// SIMATIC S7-200 project (STEP 7-Micro/WIN), CPU 224 CN REL 02.01

// OB1: protected block, not included

SUBROUTINE_BLOCK PIDCALCULATE:SBR0
TITLE=子程序注释
BEGIN
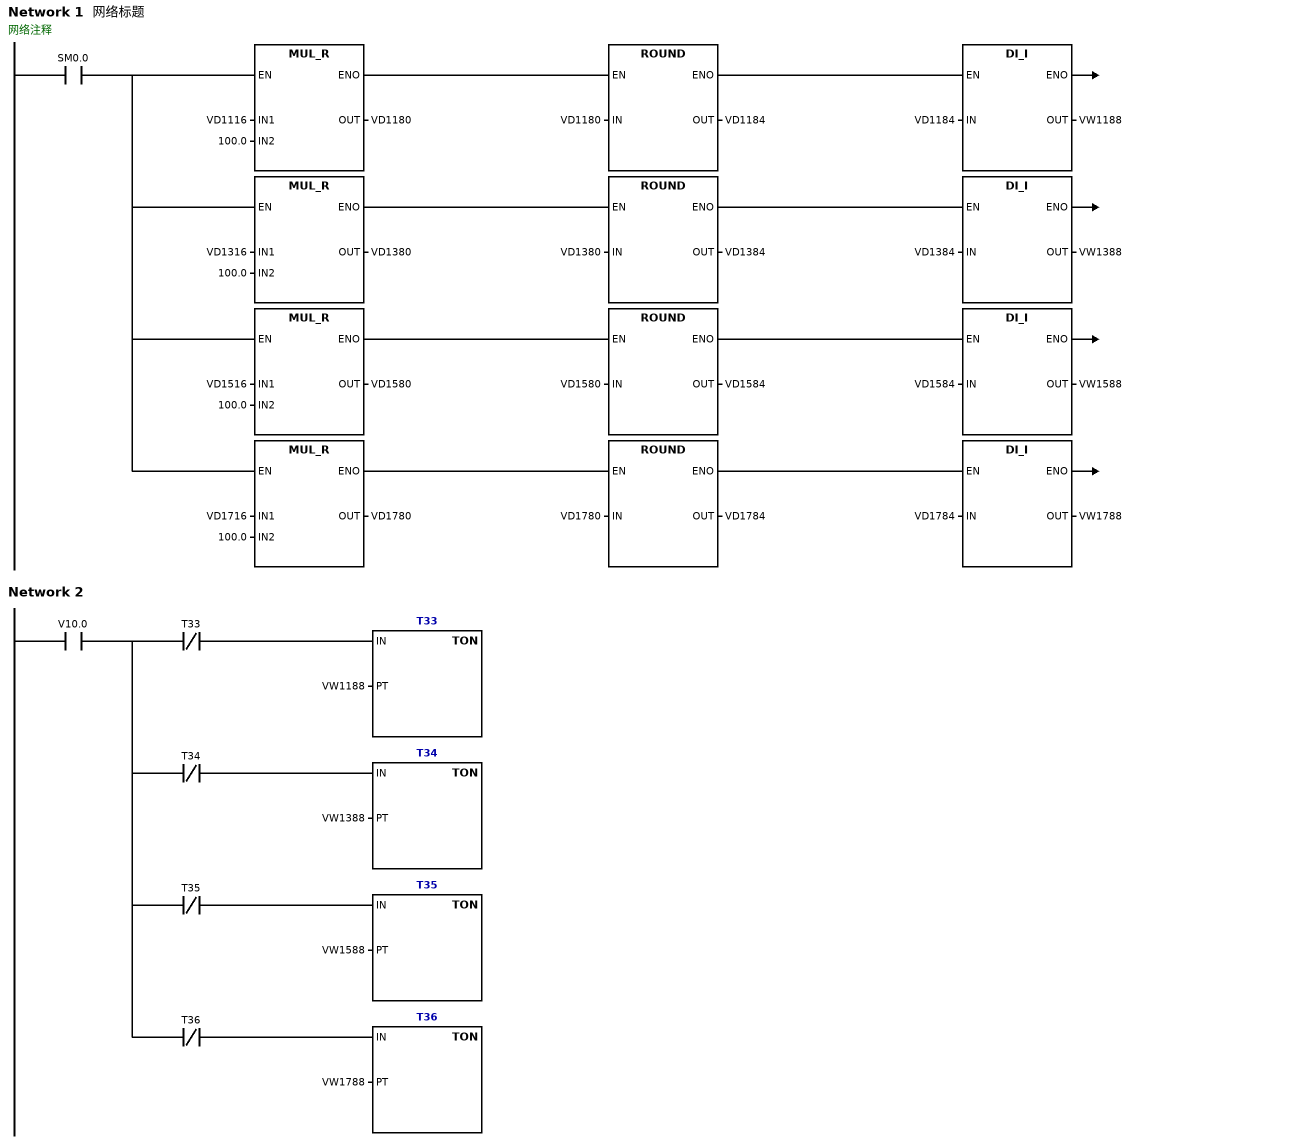
Network 1 // 网络标题
// 网络注释
LD     SM0.0
LPS
MOVR   VD1116, VD1180
AENO
*R     100.0, VD1180
AENO
ROUND  VD1180, VD1184
AENO
DTI    VD1184, VW1188
LRD
MOVR   VD1316, VD1380
AENO
*R     100.0, VD1380
AENO
ROUND  VD1380, VD1384
AENO
DTI    VD1384, VW1388
LRD
MOVR   VD1516, VD1580
AENO
*R     100.0, VD1580
AENO
ROUND  VD1580, VD1584
AENO
DTI    VD1584, VW1588
LPP
MOVR   VD1716, VD1780
AENO
*R     100.0, VD1780
AENO
ROUND  VD1780, VD1784
AENO
DTI    VD1784, VW1788
Network 2
LD     V10.0
LPS
AN     T33
TON    T33, VW1188
LRD
AN     T34
TON    T34, VW1388
LRD
AN     T35
TON    T35, VW1588
LPP
AN     T36
TON    T36, VW1788
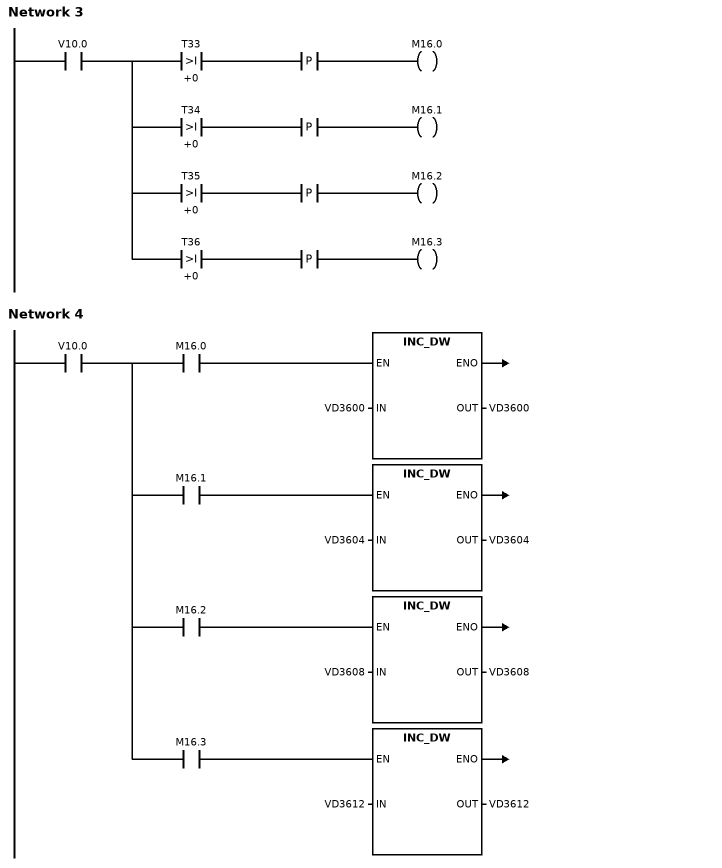
Network 3
LD     V10.0
LPS
AW>    T33, +0
EU
=      M16.0
LRD
AW>    T34, +0
EU
=      M16.1
LRD
AW>    T35, +0
EU
=      M16.2
LPP
AW>    T36, +0
EU
=      M16.3
Network 4
LD     V10.0
LPS
A      M16.0
INCD   VD3600
LRD
A      M16.1
INCD   VD3604
LRD
A      M16.2
INCD   VD3608
LPP
A      M16.3
INCD   VD3612
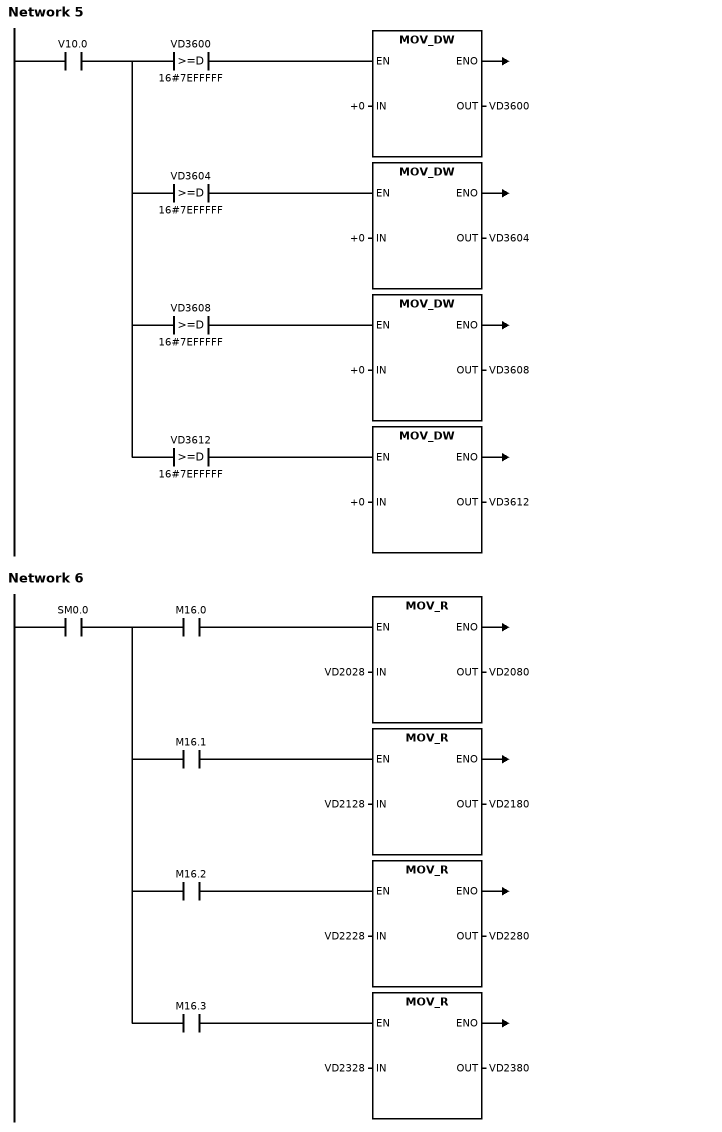
Network 5
LD     V10.0
LPS
AD>=   VD3600, 16#7EFFFFF
MOVD   +0, VD3600
LRD
AD>=   VD3604, 16#7EFFFFF
MOVD   +0, VD3604
LRD
AD>=   VD3608, 16#7EFFFFF
MOVD   +0, VD3608
LPP
AD>=   VD3612, 16#7EFFFFF
MOVD   +0, VD3612
Network 6
LD     SM0.0
LPS
A      M16.0
MOVR   VD2028, VD2080
LRD
A      M16.1
MOVR   VD2128, VD2180
LRD
A      M16.2
MOVR   VD2228, VD2280
LPP
A      M16.3
MOVR   VD2328, VD2380
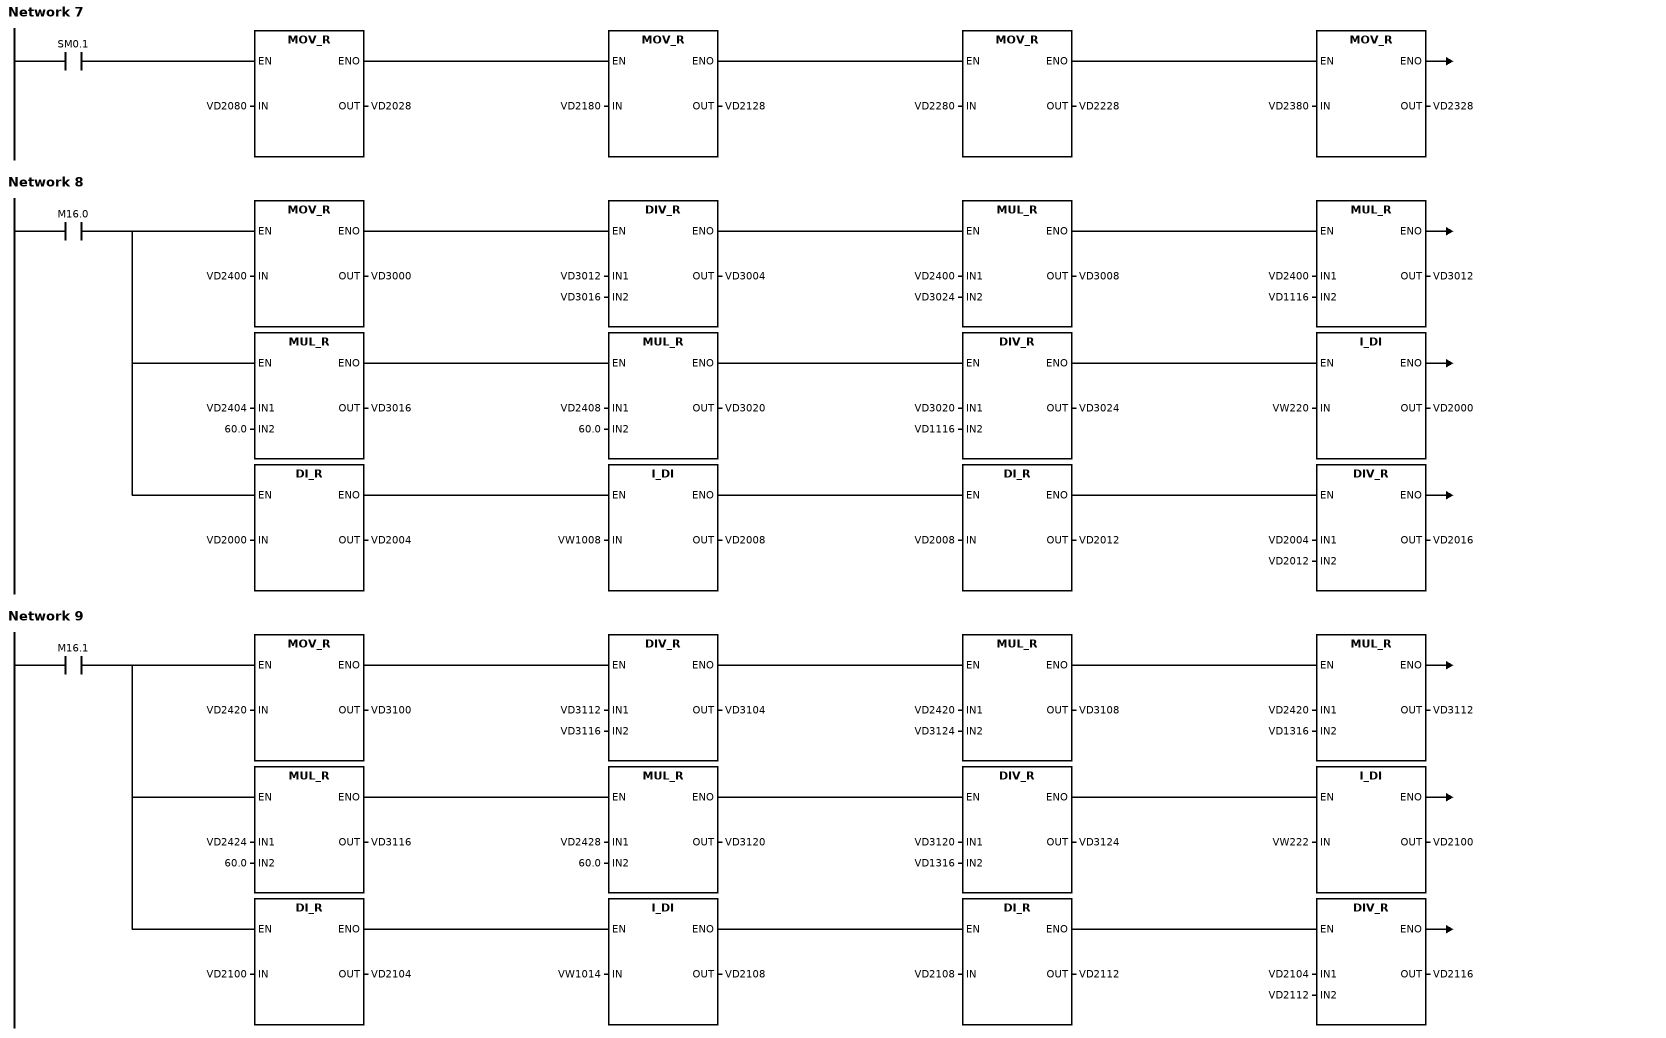
Network 7
LD     SM0.1
MOVR   VD2080, VD2028
AENO
MOVR   VD2180, VD2128
AENO
MOVR   VD2280, VD2228
AENO
MOVR   VD2380, VD2328
Network 8
LD     M16.0
LPS
MOVR   VD2400, VD3000
AENO
MOVR   VD3012, VD3004
AENO
/R     VD3016, VD3004
AENO
MOVR   VD2400, VD3008
AENO
*R     VD3024, VD3008
AENO
MOVR   VD2400, VD3012
*R     VD1116, VD3012
LRD
MOVR   VD2404, VD3016
AENO
*R     60.0, VD3016
AENO
MOVR   VD2408, VD3020
AENO
*R     60.0, VD3020
AENO
MOVR   VD3020, VD3024
AENO
/R     VD1116, VD3024
AENO
ITD    VW220, VD2000
LPP
DTR    VD2000, VD2004
AENO
ITD    VW1008, VD2008
AENO
DTR    VD2008, VD2012
AENO
MOVR   VD2004, VD2016
/R     VD2012, VD2016
Network 9
LD     M16.1
LPS
MOVR   VD2420, VD3100
AENO
MOVR   VD3112, VD3104
AENO
/R     VD3116, VD3104
AENO
MOVR   VD2420, VD3108
AENO
*R     VD3124, VD3108
AENO
MOVR   VD2420, VD3112
*R     VD1316, VD3112
LRD
MOVR   VD2424, VD3116
AENO
*R     60.0, VD3116
AENO
MOVR   VD2428, VD3120
AENO
*R     60.0, VD3120
AENO
MOVR   VD3120, VD3124
AENO
/R     VD1316, VD3124
AENO
ITD    VW222, VD2100
LPP
DTR    VD2100, VD2104
AENO
ITD    VW1014, VD2108
AENO
DTR    VD2108, VD2112
AENO
MOVR   VD2104, VD2116
/R     VD2112, VD2116
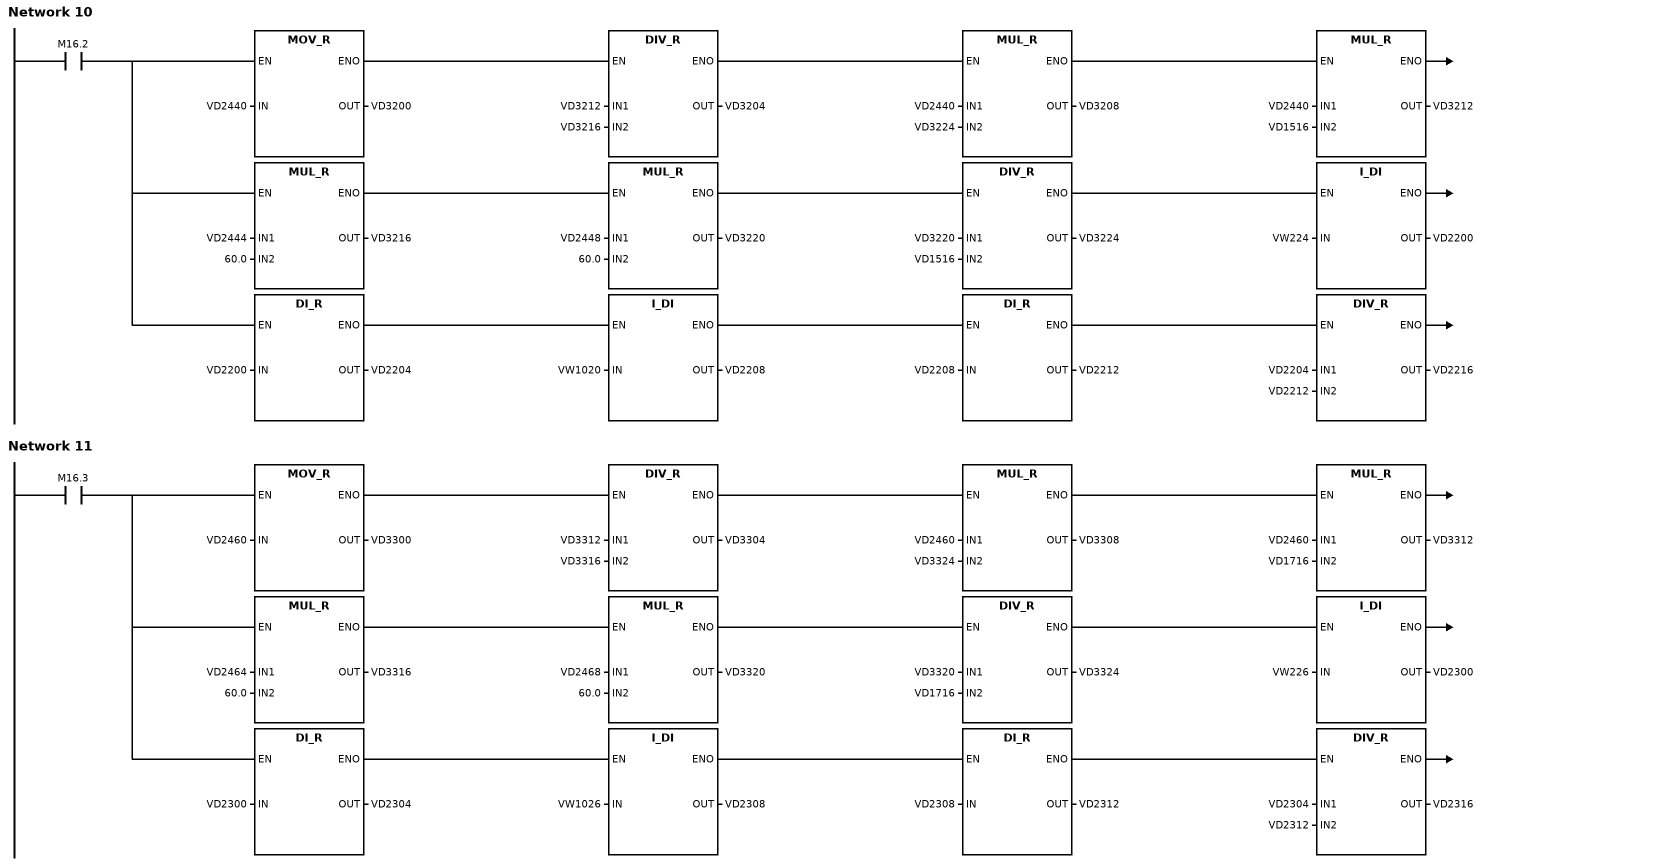
Network 10
LD     M16.2
LPS
MOVR   VD2440, VD3200
AENO
MOVR   VD3212, VD3204
AENO
/R     VD3216, VD3204
AENO
MOVR   VD2440, VD3208
AENO
*R     VD3224, VD3208
AENO
MOVR   VD2440, VD3212
*R     VD1516, VD3212
LRD
MOVR   VD2444, VD3216
AENO
*R     60.0, VD3216
AENO
MOVR   VD2448, VD3220
AENO
*R     60.0, VD3220
AENO
MOVR   VD3220, VD3224
AENO
/R     VD1516, VD3224
AENO
ITD    VW224, VD2200
LPP
DTR    VD2200, VD2204
AENO
ITD    VW1020, VD2208
AENO
DTR    VD2208, VD2212
AENO
MOVR   VD2204, VD2216
/R     VD2212, VD2216
Network 11
LD     M16.3
LPS
MOVR   VD2460, VD3300
AENO
MOVR   VD3312, VD3304
AENO
/R     VD3316, VD3304
AENO
MOVR   VD2460, VD3308
AENO
*R     VD3324, VD3308
AENO
MOVR   VD2460, VD3312
*R     VD1716, VD3312
LRD
MOVR   VD2464, VD3316
AENO
*R     60.0, VD3316
AENO
MOVR   VD2468, VD3320
AENO
*R     60.0, VD3320
AENO
MOVR   VD3320, VD3324
AENO
/R     VD1716, VD3324
AENO
ITD    VW226, VD2300
LPP
DTR    VD2300, VD2304
AENO
ITD    VW1026, VD2308
AENO
DTR    VD2308, VD2312
AENO
MOVR   VD2304, VD2316
/R     VD2312, VD2316
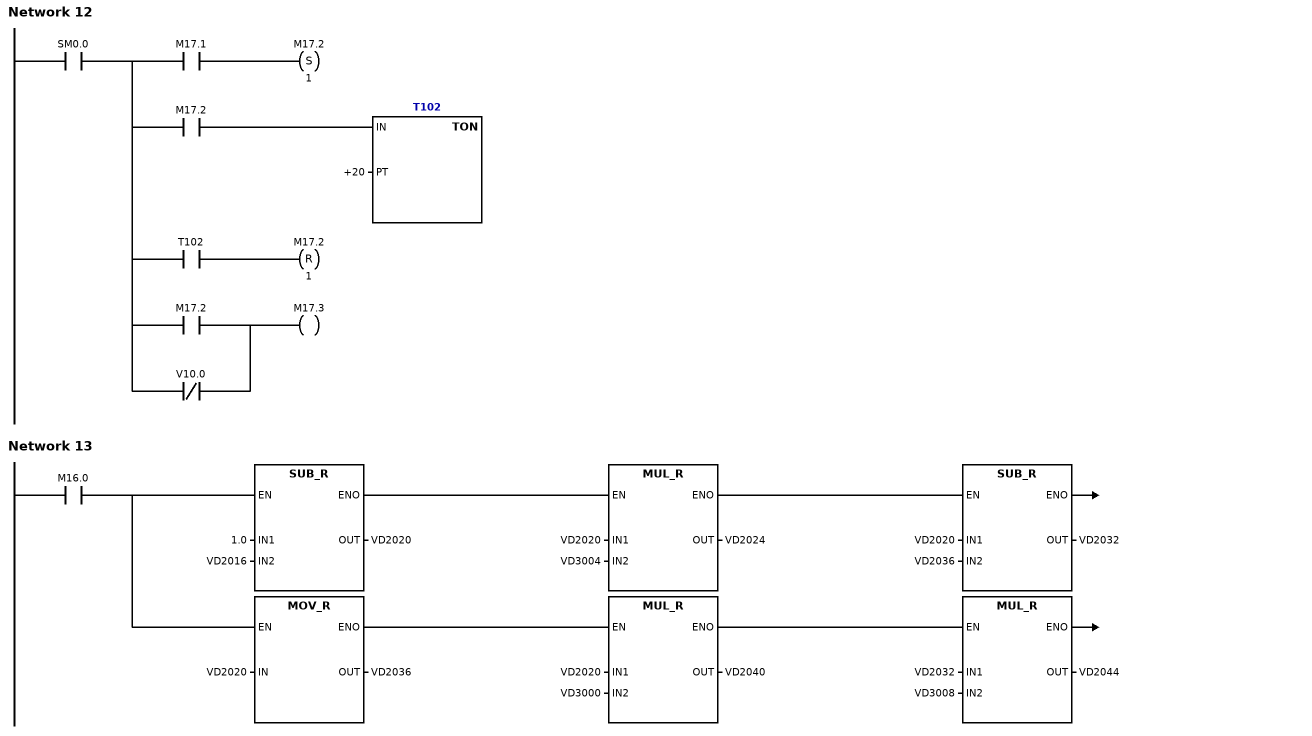
Network 12
LD     SM0.0
LPS
A      M17.1
S      M17.2, 1
LRD
A      M17.2
TON    T102, +20
LRD
A      T102
R      M17.2, 1
LPP
LD     M17.2
ON     V10.0
ALD
=      M17.3
Network 13
LD     M16.0
LPS
MOVR   1.0, VD2020
AENO
-R     VD2016, VD2020
AENO
MOVR   VD2020, VD2024
AENO
*R     VD3004, VD2024
AENO
MOVR   VD2020, VD2032
-R     VD2036, VD2032
LPP
MOVR   VD2020, VD2036
AENO
MOVR   VD2020, VD2040
AENO
*R     VD3000, VD2040
AENO
MOVR   VD2032, VD2044
*R     VD3008, VD2044
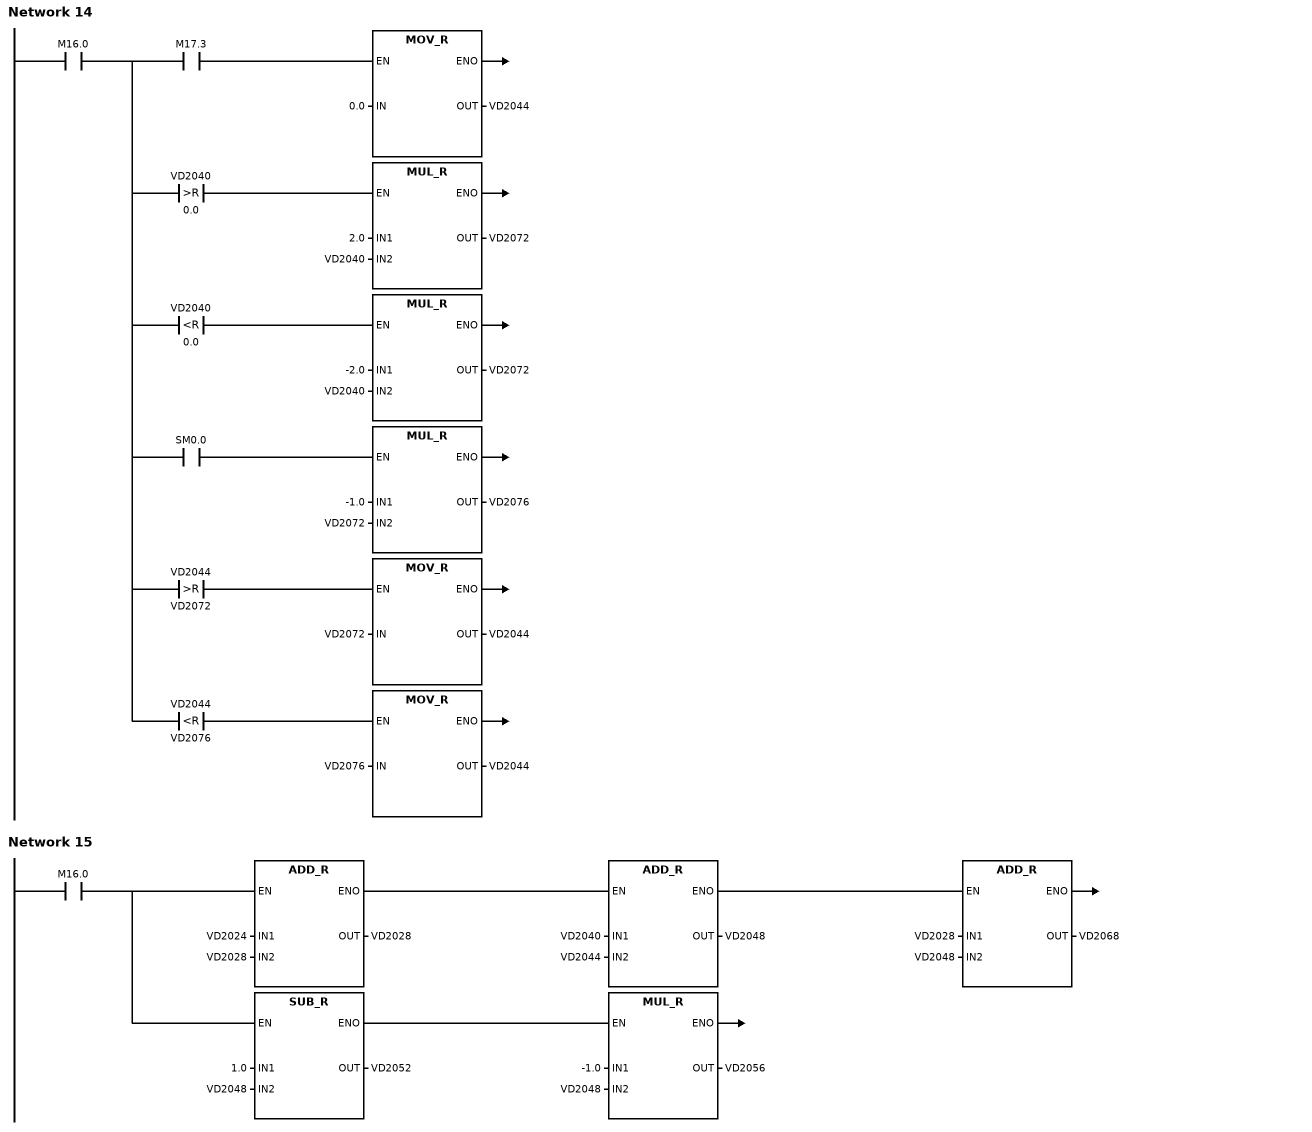
Network 14
LD     M16.0
LPS
A      M17.3
MOVR   0.0, VD2044
LRD
AR>    VD2040, 0.0
MOVR   2.0, VD2072
*R     VD2040, VD2072
LRD
AR<    VD2040, 0.0
MOVR   -2.0, VD2072
*R     VD2040, VD2072
LRD
A      SM0.0
MOVR   -1.0, VD2076
*R     VD2072, VD2076
LRD
AR>    VD2044, VD2072
MOVR   VD2072, VD2044
LPP
AR<    VD2044, VD2076
MOVR   VD2076, VD2044
Network 15
LD     M16.0
LPS
+R     VD2024, VD2028
AENO
MOVR   VD2040, VD2048
AENO
+R     VD2044, VD2048
AENO
MOVR   VD2028, VD2068
+R     VD2048, VD2068
LPP
MOVR   1.0, VD2052
AENO
-R     VD2048, VD2052
AENO
MOVR   -1.0, VD2056
*R     VD2048, VD2056
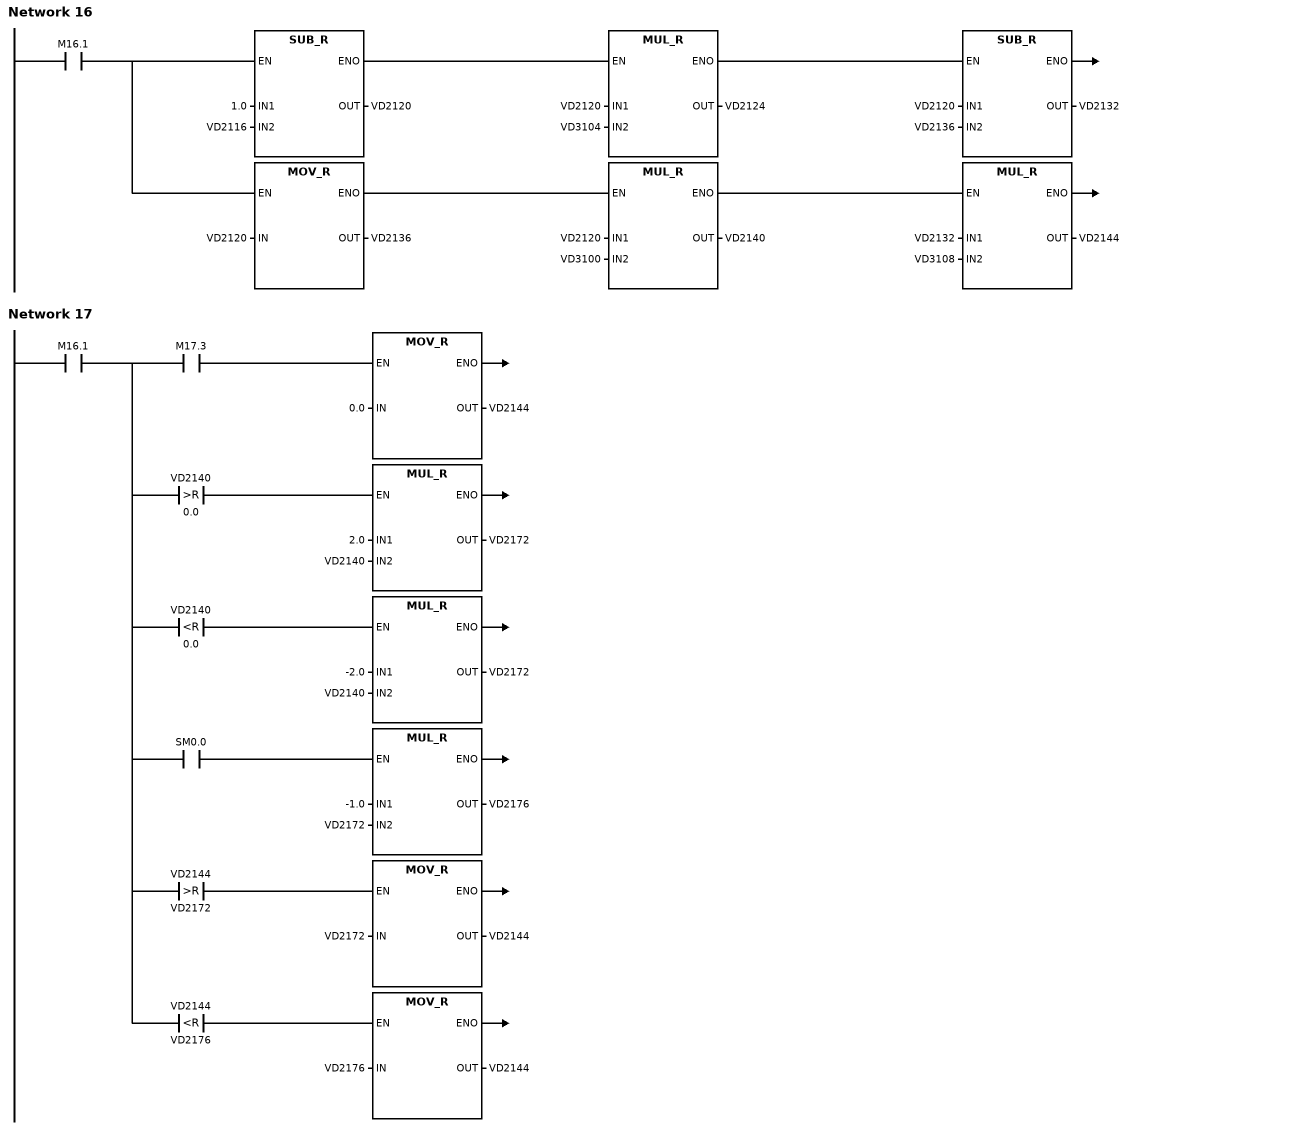
Network 16
LD     M16.1
LPS
MOVR   1.0, VD2120
AENO
-R     VD2116, VD2120
AENO
MOVR   VD2120, VD2124
AENO
*R     VD3104, VD2124
AENO
MOVR   VD2120, VD2132
-R     VD2136, VD2132
LPP
MOVR   VD2120, VD2136
AENO
MOVR   VD2120, VD2140
AENO
*R     VD3100, VD2140
AENO
MOVR   VD2132, VD2144
*R     VD3108, VD2144
Network 17
LD     M16.1
LPS
A      M17.3
MOVR   0.0, VD2144
LRD
AR>    VD2140, 0.0
MOVR   2.0, VD2172
*R     VD2140, VD2172
LRD
AR<    VD2140, 0.0
MOVR   -2.0, VD2172
*R     VD2140, VD2172
LRD
A      SM0.0
MOVR   -1.0, VD2176
*R     VD2172, VD2176
LRD
AR>    VD2144, VD2172
MOVR   VD2172, VD2144
LPP
AR<    VD2144, VD2176
MOVR   VD2176, VD2144
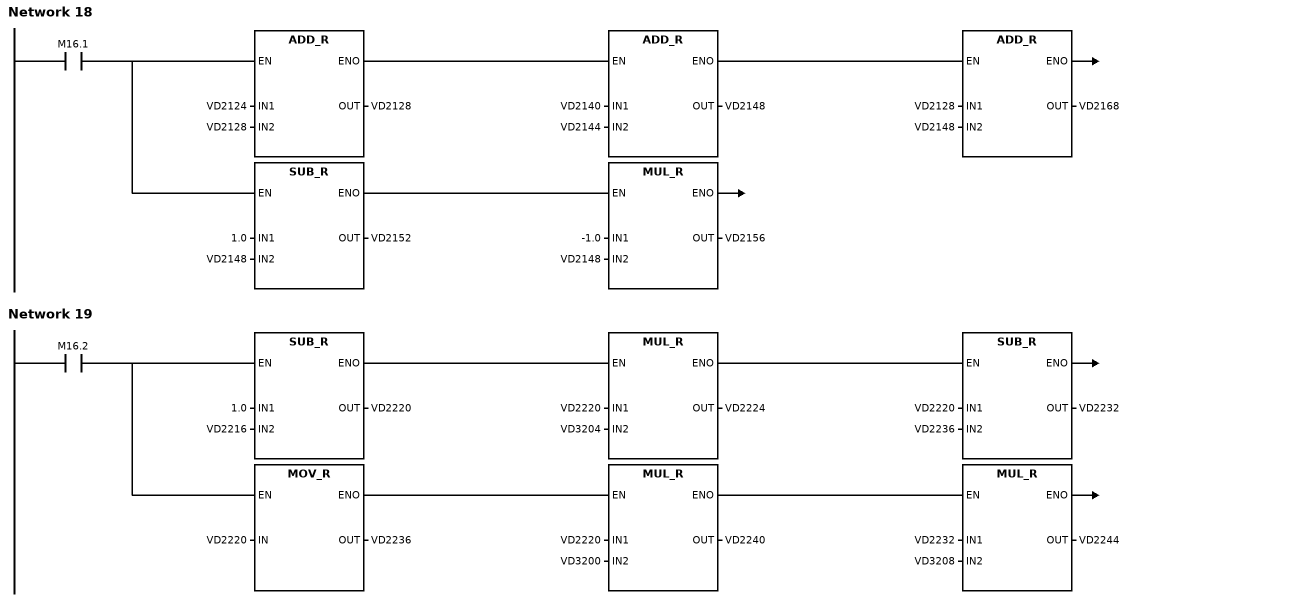
Network 18
LD     M16.1
LPS
+R     VD2124, VD2128
AENO
MOVR   VD2140, VD2148
AENO
+R     VD2144, VD2148
AENO
MOVR   VD2128, VD2168
+R     VD2148, VD2168
LPP
MOVR   1.0, VD2152
AENO
-R     VD2148, VD2152
AENO
MOVR   -1.0, VD2156
*R     VD2148, VD2156
Network 19
LD     M16.2
LPS
MOVR   1.0, VD2220
AENO
-R     VD2216, VD2220
AENO
MOVR   VD2220, VD2224
AENO
*R     VD3204, VD2224
AENO
MOVR   VD2220, VD2232
-R     VD2236, VD2232
LPP
MOVR   VD2220, VD2236
AENO
MOVR   VD2220, VD2240
AENO
*R     VD3200, VD2240
AENO
MOVR   VD2232, VD2244
*R     VD3208, VD2244
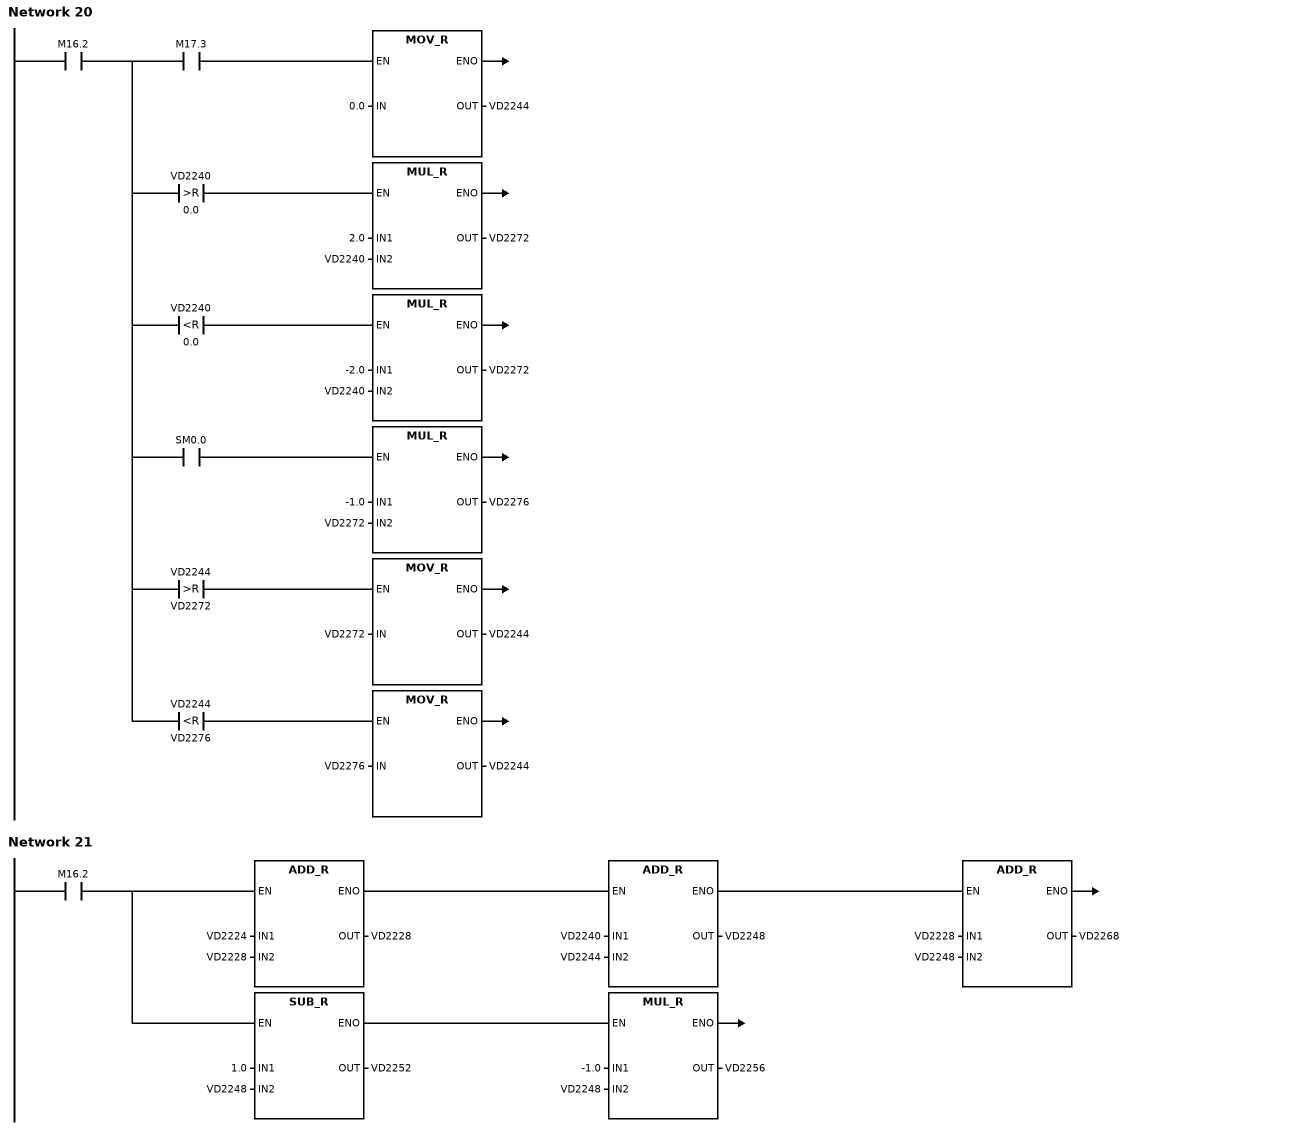
Network 20
LD     M16.2
LPS
A      M17.3
MOVR   0.0, VD2244
LRD
AR>    VD2240, 0.0
MOVR   2.0, VD2272
*R     VD2240, VD2272
LRD
AR<    VD2240, 0.0
MOVR   -2.0, VD2272
*R     VD2240, VD2272
LRD
A      SM0.0
MOVR   -1.0, VD2276
*R     VD2272, VD2276
LRD
AR>    VD2244, VD2272
MOVR   VD2272, VD2244
LPP
AR<    VD2244, VD2276
MOVR   VD2276, VD2244
Network 21
LD     M16.2
LPS
+R     VD2224, VD2228
AENO
MOVR   VD2240, VD2248
AENO
+R     VD2244, VD2248
AENO
MOVR   VD2228, VD2268
+R     VD2248, VD2268
LPP
MOVR   1.0, VD2252
AENO
-R     VD2248, VD2252
AENO
MOVR   -1.0, VD2256
*R     VD2248, VD2256
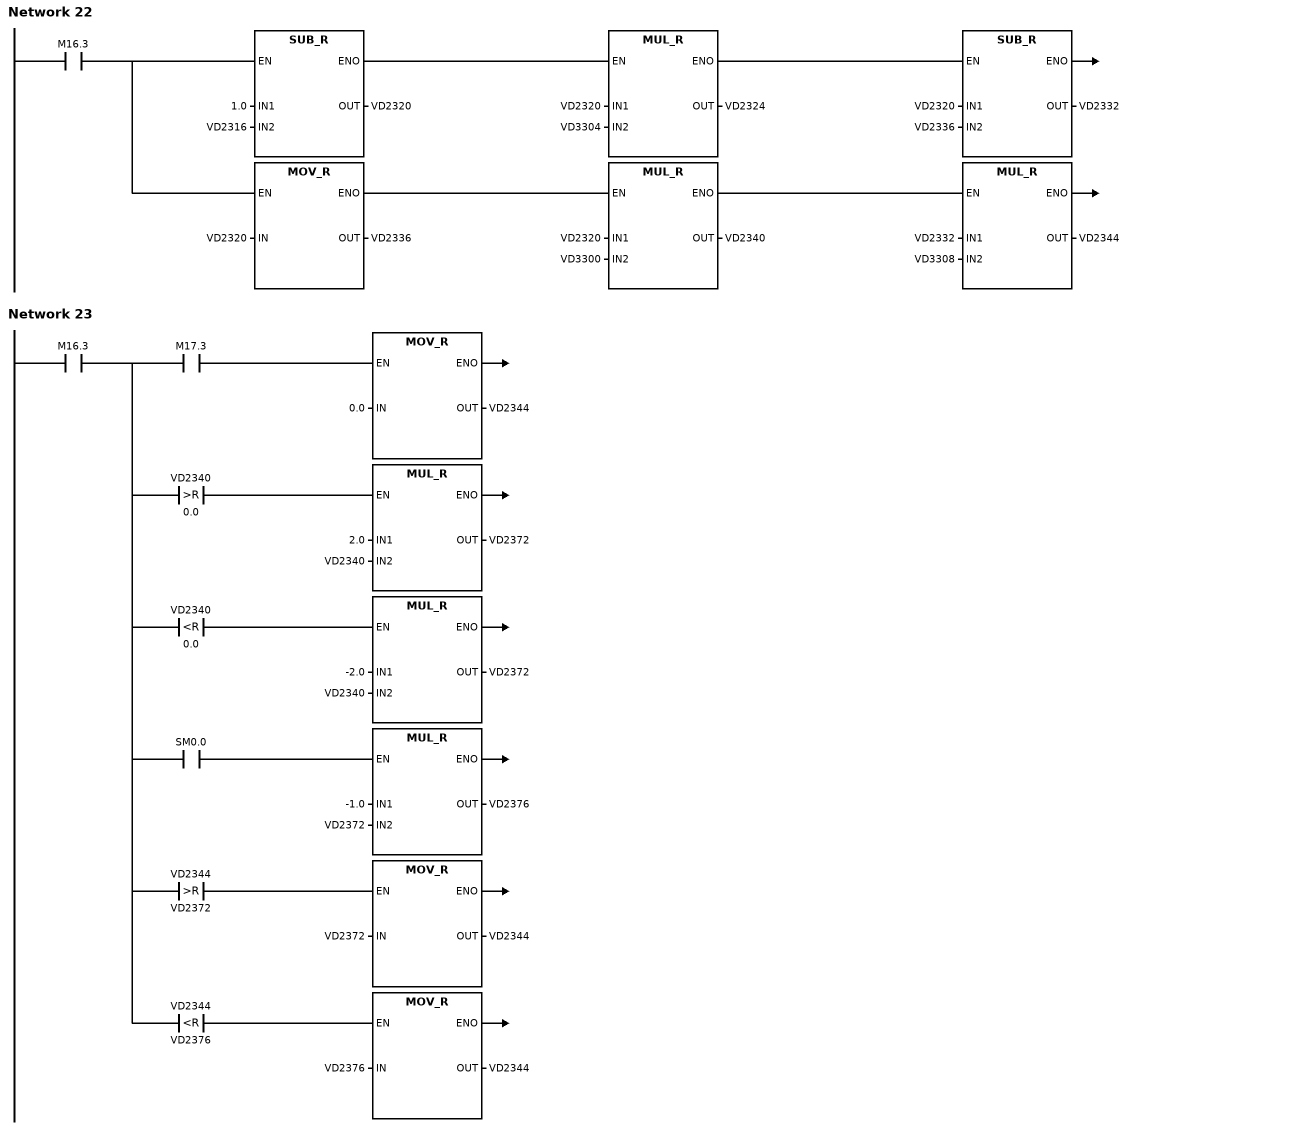
Network 22
LD     M16.3
LPS
MOVR   1.0, VD2320
AENO
-R     VD2316, VD2320
AENO
MOVR   VD2320, VD2324
AENO
*R     VD3304, VD2324
AENO
MOVR   VD2320, VD2332
-R     VD2336, VD2332
LPP
MOVR   VD2320, VD2336
AENO
MOVR   VD2320, VD2340
AENO
*R     VD3300, VD2340
AENO
MOVR   VD2332, VD2344
*R     VD3308, VD2344
Network 23
LD     M16.3
LPS
A      M17.3
MOVR   0.0, VD2344
LRD
AR>    VD2340, 0.0
MOVR   2.0, VD2372
*R     VD2340, VD2372
LRD
AR<    VD2340, 0.0
MOVR   -2.0, VD2372
*R     VD2340, VD2372
LRD
A      SM0.0
MOVR   -1.0, VD2376
*R     VD2372, VD2376
LRD
AR>    VD2344, VD2372
MOVR   VD2372, VD2344
LPP
AR<    VD2344, VD2376
MOVR   VD2376, VD2344
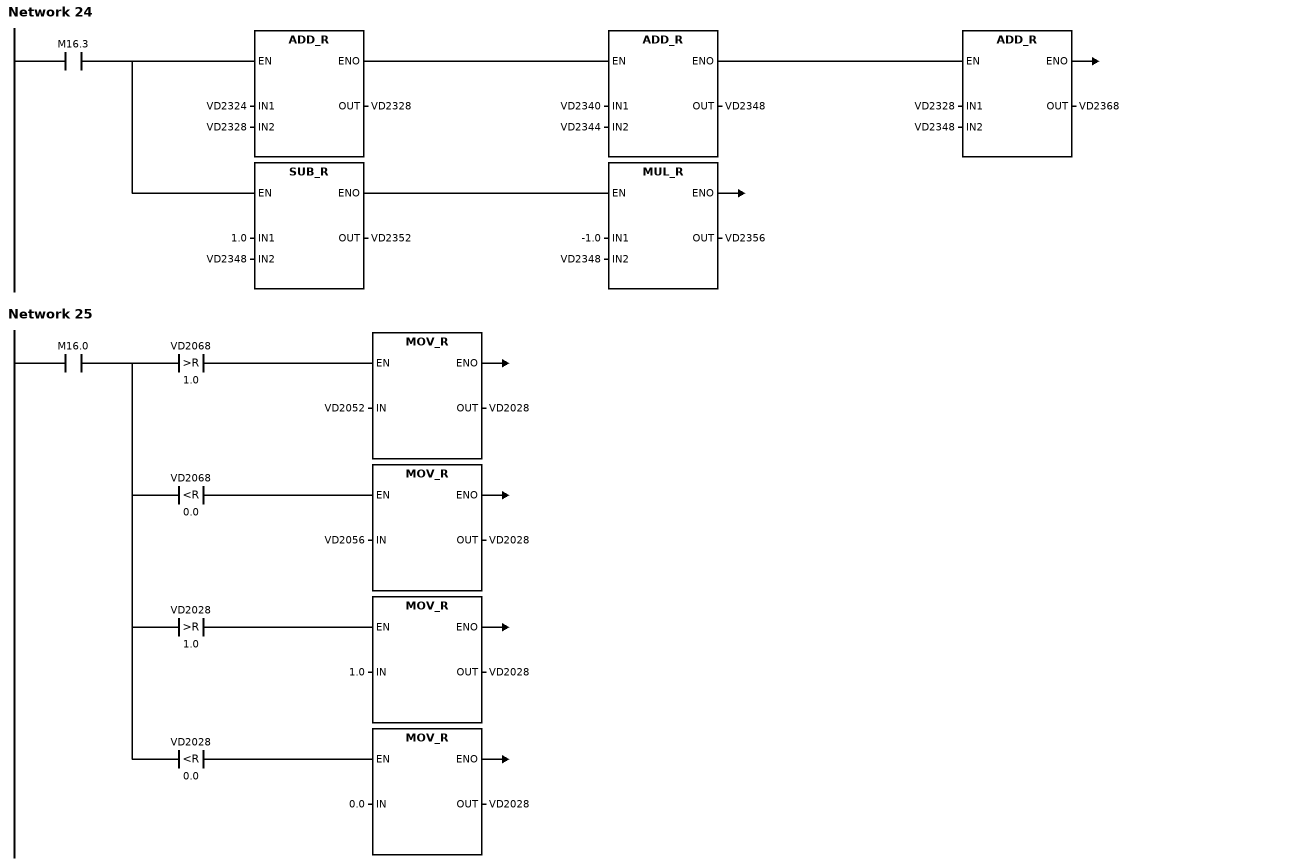
Network 24
LD     M16.3
LPS
+R     VD2324, VD2328
AENO
MOVR   VD2340, VD2348
AENO
+R     VD2344, VD2348
AENO
MOVR   VD2328, VD2368
+R     VD2348, VD2368
LPP
MOVR   1.0, VD2352
AENO
-R     VD2348, VD2352
AENO
MOVR   -1.0, VD2356
*R     VD2348, VD2356
Network 25
LD     M16.0
LPS
AR>    VD2068, 1.0
MOVR   VD2052, VD2028
LRD
AR<    VD2068, 0.0
MOVR   VD2056, VD2028
LRD
AR>    VD2028, 1.0
MOVR   1.0, VD2028
LPP
AR<    VD2028, 0.0
MOVR   0.0, VD2028
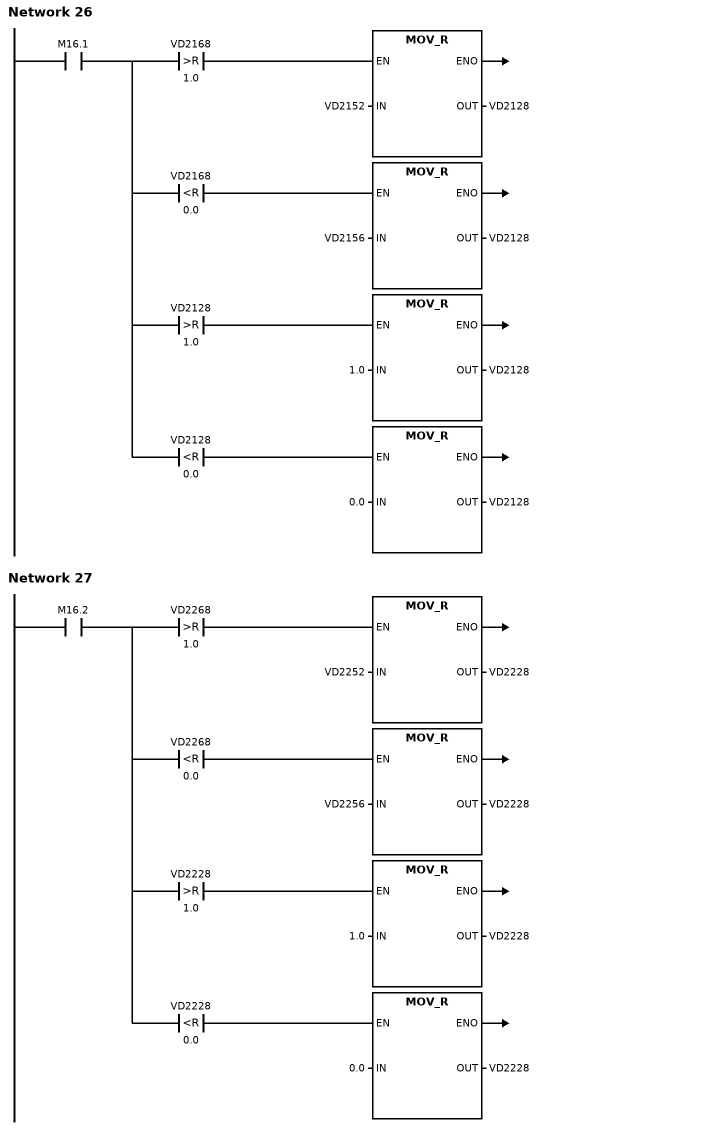
Network 26
LD     M16.1
LPS
AR>    VD2168, 1.0
MOVR   VD2152, VD2128
LRD
AR<    VD2168, 0.0
MOVR   VD2156, VD2128
LRD
AR>    VD2128, 1.0
MOVR   1.0, VD2128
LPP
AR<    VD2128, 0.0
MOVR   0.0, VD2128
Network 27
LD     M16.2
LPS
AR>    VD2268, 1.0
MOVR   VD2252, VD2228
LRD
AR<    VD2268, 0.0
MOVR   VD2256, VD2228
LRD
AR>    VD2228, 1.0
MOVR   1.0, VD2228
LPP
AR<    VD2228, 0.0
MOVR   0.0, VD2228
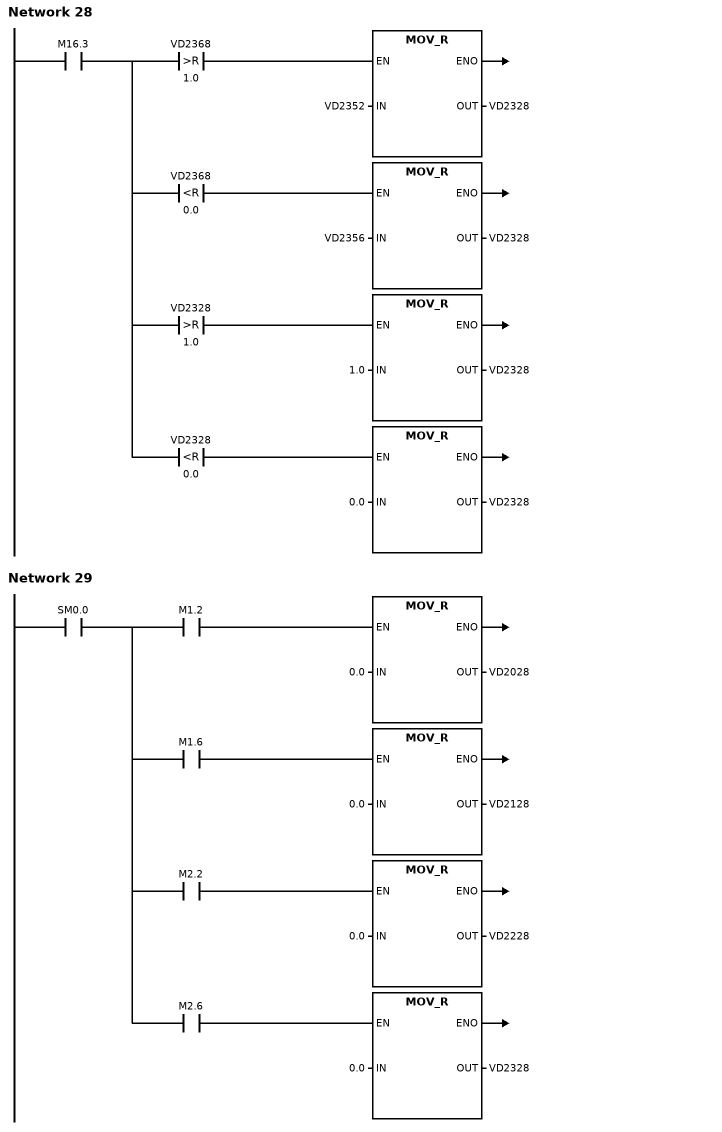
Network 28
LD     M16.3
LPS
AR>    VD2368, 1.0
MOVR   VD2352, VD2328
LRD
AR<    VD2368, 0.0
MOVR   VD2356, VD2328
LRD
AR>    VD2328, 1.0
MOVR   1.0, VD2328
LPP
AR<    VD2328, 0.0
MOVR   0.0, VD2328
Network 29
LD     SM0.0
LPS
A      M1.2
MOVR   0.0, VD2028
LRD
A      M1.6
MOVR   0.0, VD2128
LRD
A      M2.2
MOVR   0.0, VD2228
LPP
A      M2.6
MOVR   0.0, VD2328
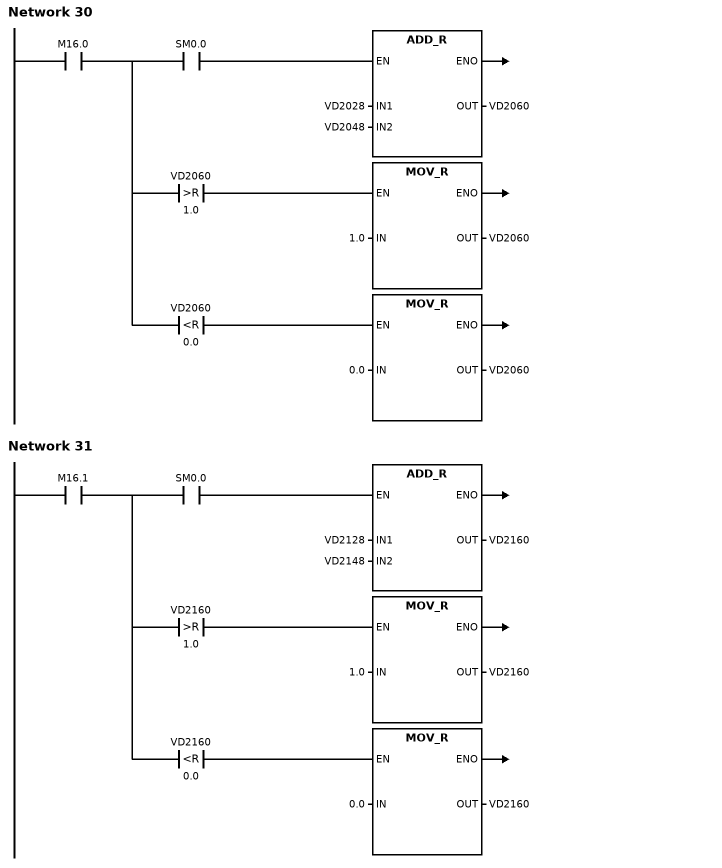
Network 30
LD     M16.0
LPS
A      SM0.0
MOVR   VD2028, VD2060
+R     VD2048, VD2060
LRD
AR>    VD2060, 1.0
MOVR   1.0, VD2060
LPP
AR<    VD2060, 0.0
MOVR   0.0, VD2060
Network 31
LD     M16.1
LPS
A      SM0.0
MOVR   VD2128, VD2160
+R     VD2148, VD2160
LRD
AR>    VD2160, 1.0
MOVR   1.0, VD2160
LPP
AR<    VD2160, 0.0
MOVR   0.0, VD2160
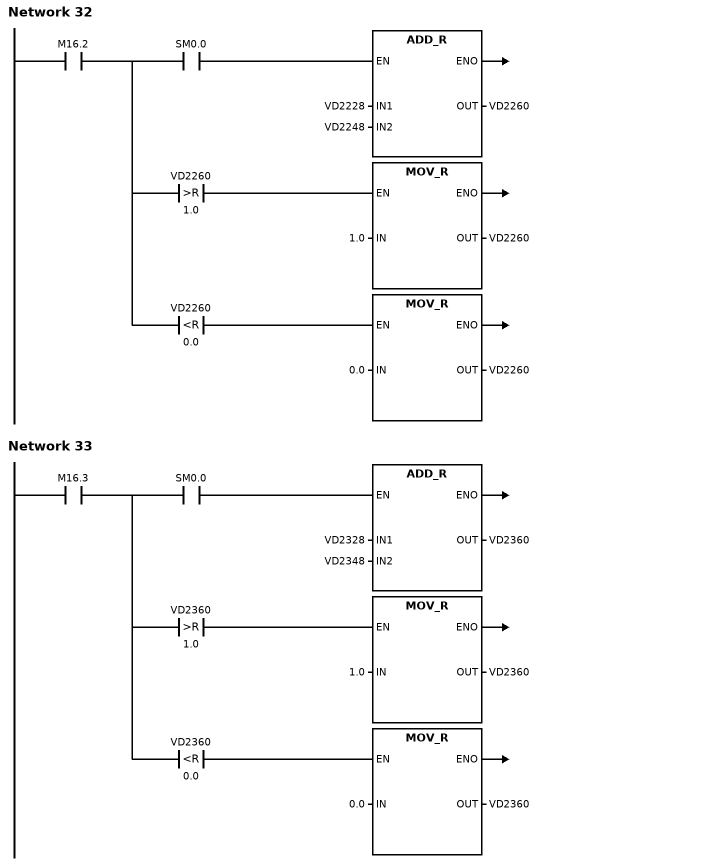
Network 32
LD     M16.2
LPS
A      SM0.0
MOVR   VD2228, VD2260
+R     VD2248, VD2260
LRD
AR>    VD2260, 1.0
MOVR   1.0, VD2260
LPP
AR<    VD2260, 0.0
MOVR   0.0, VD2260
Network 33
LD     M16.3
LPS
A      SM0.0
MOVR   VD2328, VD2360
+R     VD2348, VD2360
LRD
AR>    VD2360, 1.0
MOVR   1.0, VD2360
LPP
AR<    VD2360, 0.0
MOVR   0.0, VD2360
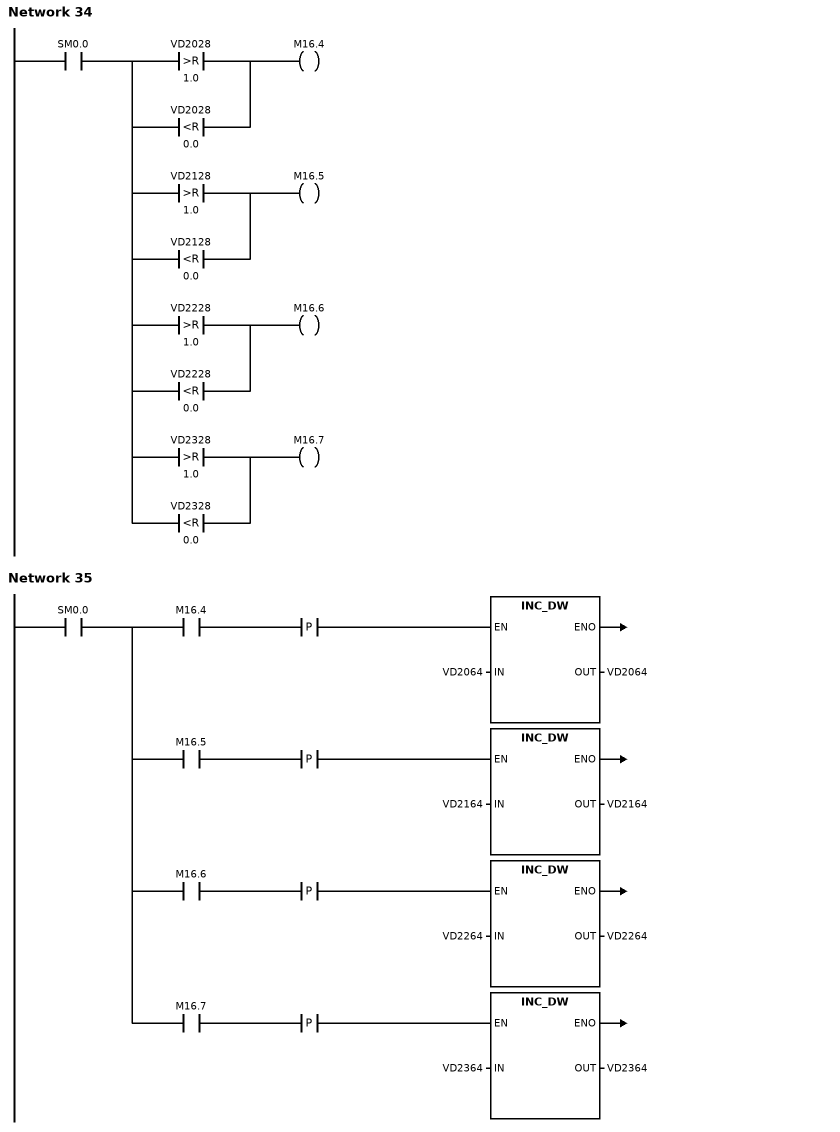
Network 34
LD     SM0.0
LPS
LDR>   VD2028, 1.0
OR<    VD2028, 0.0
ALD
=      M16.4
LRD
LDR>   VD2128, 1.0
OR<    VD2128, 0.0
ALD
=      M16.5
LRD
LDR>   VD2228, 1.0
OR<    VD2228, 0.0
ALD
=      M16.6
LPP
LDR>   VD2328, 1.0
OR<    VD2328, 0.0
ALD
=      M16.7
Network 35
LD     SM0.0
LPS
A      M16.4
EU
INCD   VD2064
LRD
A      M16.5
EU
INCD   VD2164
LRD
A      M16.6
EU
INCD   VD2264
LPP
A      M16.7
EU
INCD   VD2364
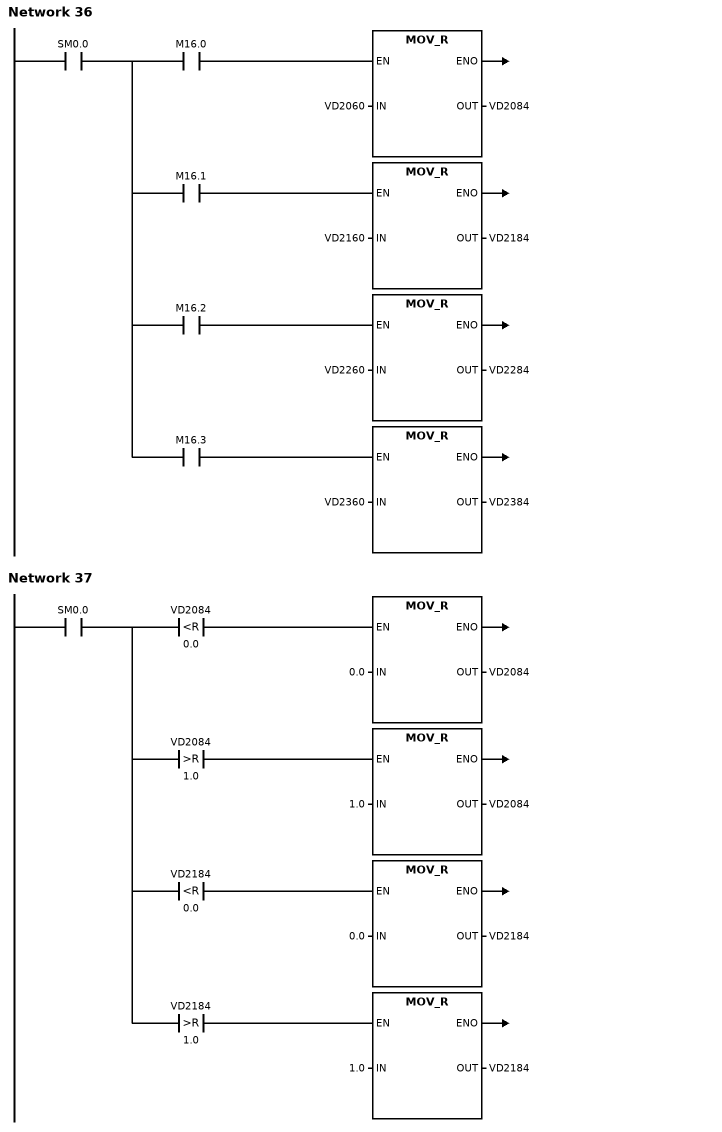
Network 36
LD     SM0.0
LPS
A      M16.0
MOVR   VD2060, VD2084
LRD
A      M16.1
MOVR   VD2160, VD2184
LRD
A      M16.2
MOVR   VD2260, VD2284
LPP
A      M16.3
MOVR   VD2360, VD2384
Network 37
LD     SM0.0
LPS
AR<    VD2084, 0.0
MOVR   0.0, VD2084
LRD
AR>    VD2084, 1.0
MOVR   1.0, VD2084
LRD
AR<    VD2184, 0.0
MOVR   0.0, VD2184
LPP
AR>    VD2184, 1.0
MOVR   1.0, VD2184
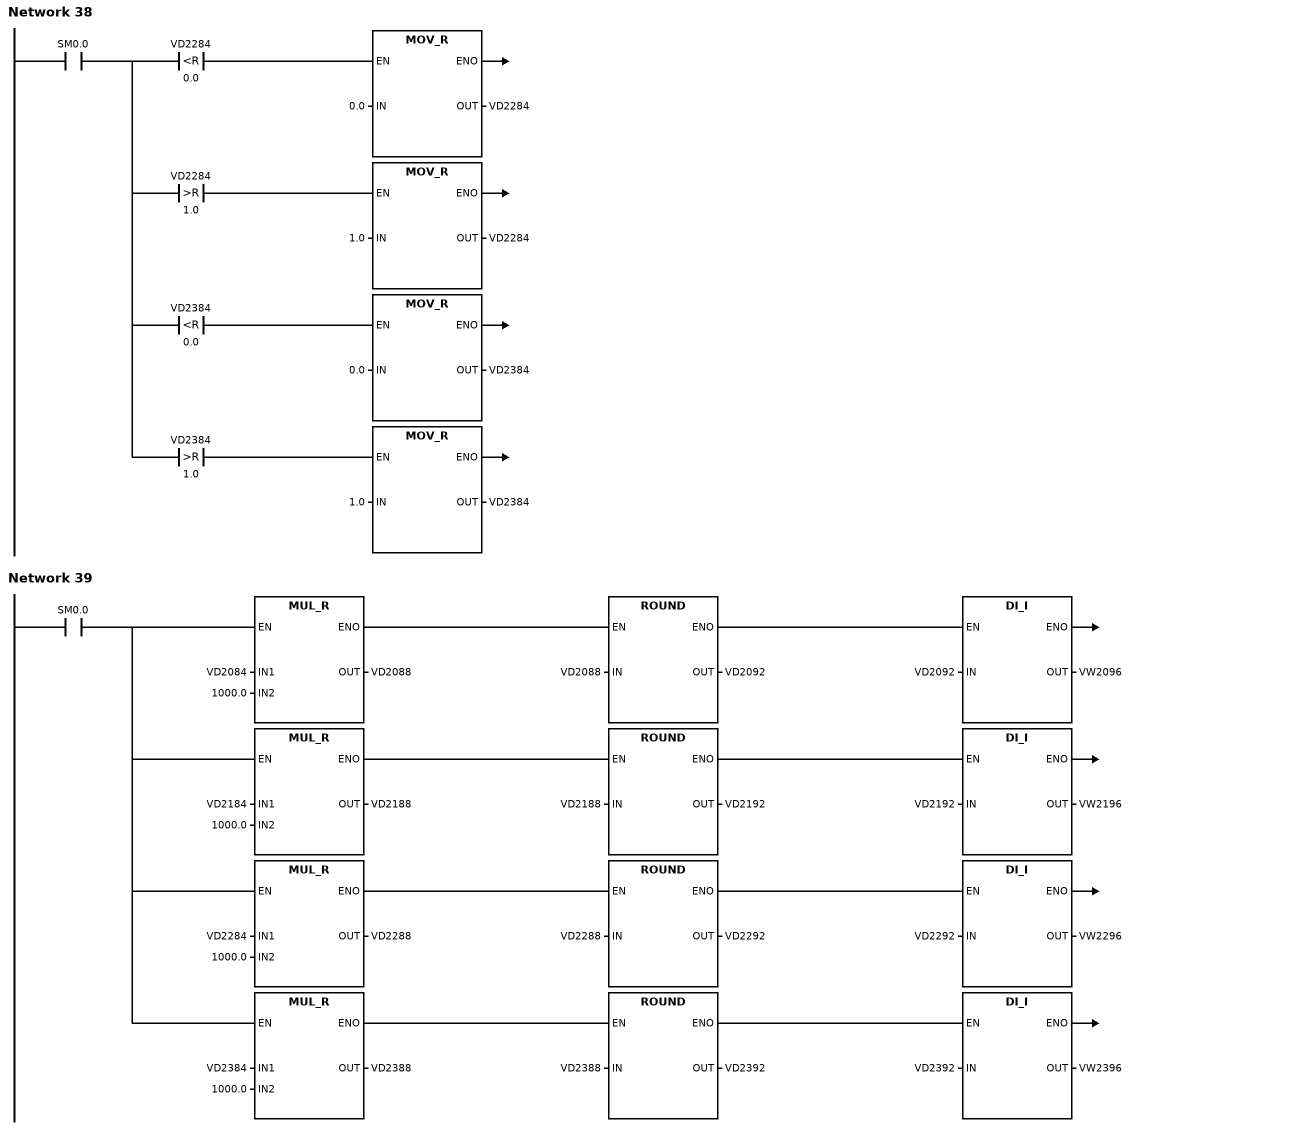
Network 38
LD     SM0.0
LPS
AR<    VD2284, 0.0
MOVR   0.0, VD2284
LRD
AR>    VD2284, 1.0
MOVR   1.0, VD2284
LRD
AR<    VD2384, 0.0
MOVR   0.0, VD2384
LPP
AR>    VD2384, 1.0
MOVR   1.0, VD2384
Network 39
LD     SM0.0
LPS
MOVR   VD2084, VD2088
AENO
*R     1000.0, VD2088
AENO
ROUND  VD2088, VD2092
AENO
DTI    VD2092, VW2096
LRD
MOVR   VD2184, VD2188
AENO
*R     1000.0, VD2188
AENO
ROUND  VD2188, VD2192
AENO
DTI    VD2192, VW2196
LRD
MOVR   VD2284, VD2288
AENO
*R     1000.0, VD2288
AENO
ROUND  VD2288, VD2292
AENO
DTI    VD2292, VW2296
LPP
MOVR   VD2384, VD2388
AENO
*R     1000.0, VD2388
AENO
ROUND  VD2388, VD2392
AENO
DTI    VD2392, VW2396
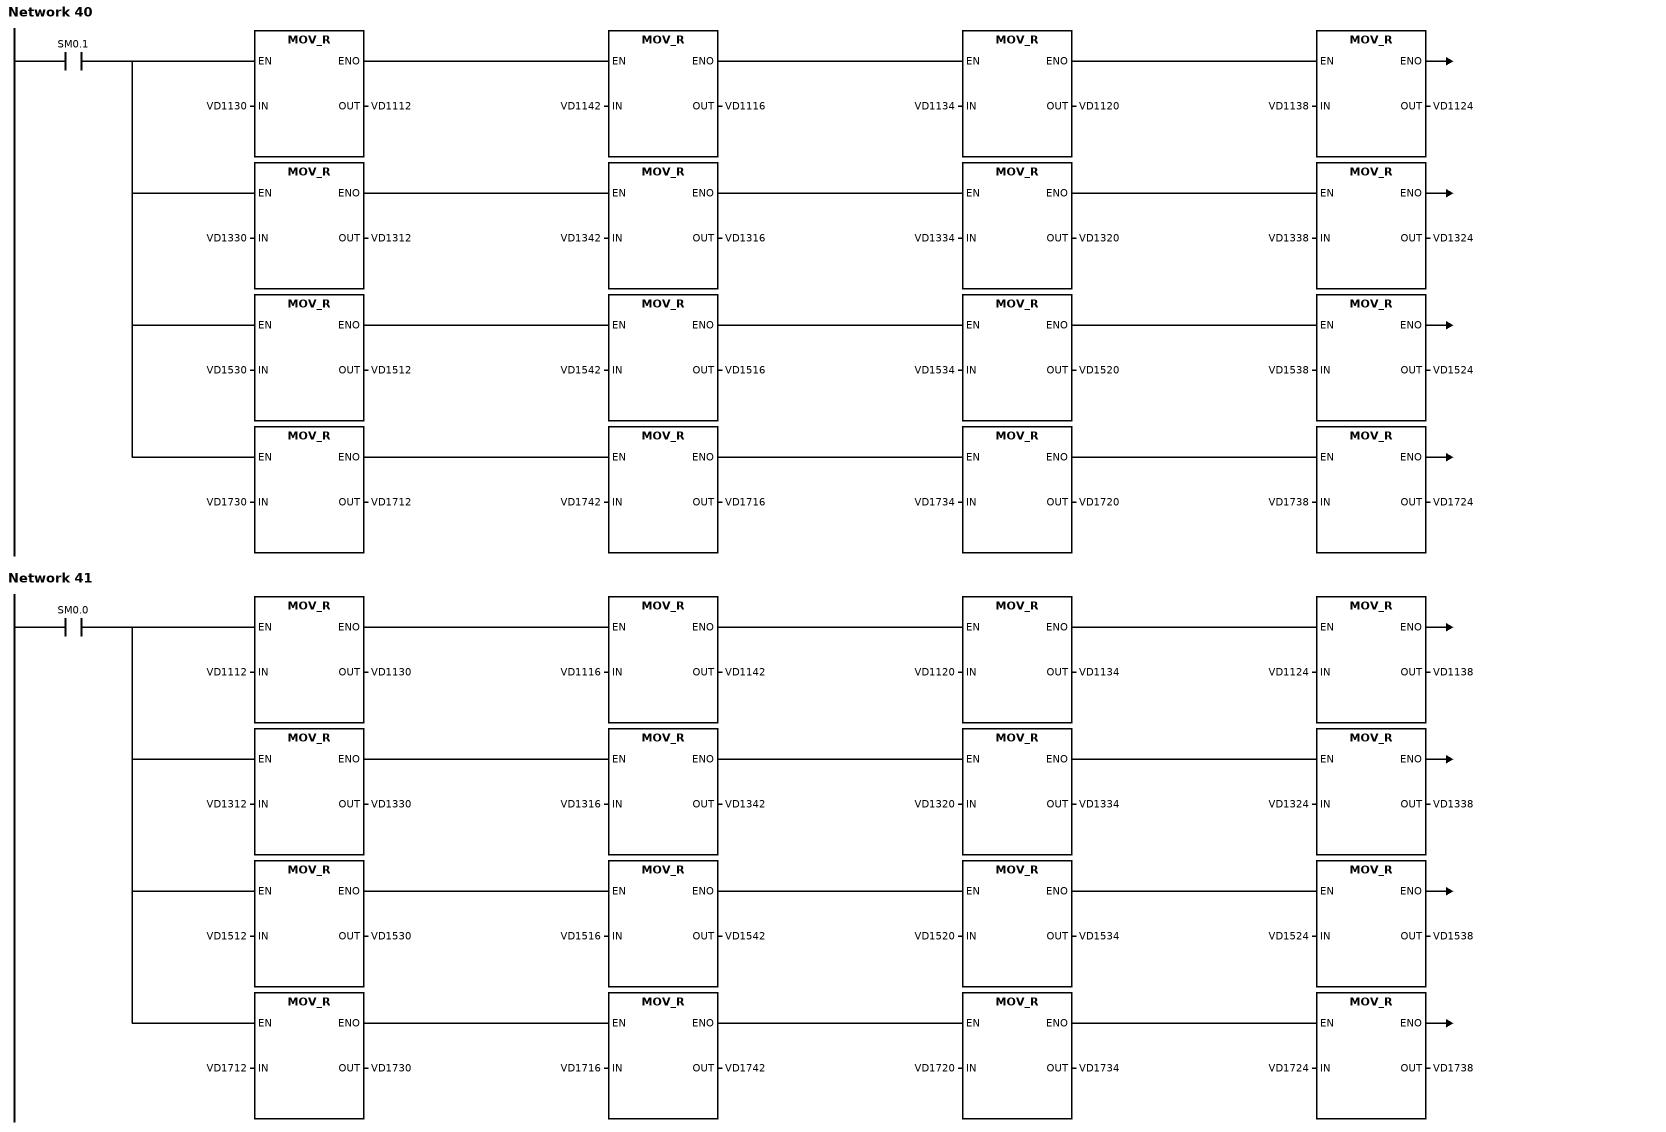
Network 40
LD     SM0.1
LPS
MOVR   VD1130, VD1112
AENO
MOVR   VD1142, VD1116
AENO
MOVR   VD1134, VD1120
AENO
MOVR   VD1138, VD1124
LRD
MOVR   VD1330, VD1312
AENO
MOVR   VD1342, VD1316
AENO
MOVR   VD1334, VD1320
AENO
MOVR   VD1338, VD1324
LRD
MOVR   VD1530, VD1512
AENO
MOVR   VD1542, VD1516
AENO
MOVR   VD1534, VD1520
AENO
MOVR   VD1538, VD1524
LPP
MOVR   VD1730, VD1712
AENO
MOVR   VD1742, VD1716
AENO
MOVR   VD1734, VD1720
AENO
MOVR   VD1738, VD1724
Network 41
LD     SM0.0
LPS
MOVR   VD1112, VD1130
AENO
MOVR   VD1116, VD1142
AENO
MOVR   VD1120, VD1134
AENO
MOVR   VD1124, VD1138
LRD
MOVR   VD1312, VD1330
AENO
MOVR   VD1316, VD1342
AENO
MOVR   VD1320, VD1334
AENO
MOVR   VD1324, VD1338
LRD
MOVR   VD1512, VD1530
AENO
MOVR   VD1516, VD1542
AENO
MOVR   VD1520, VD1534
AENO
MOVR   VD1524, VD1538
LPP
MOVR   VD1712, VD1730
AENO
MOVR   VD1716, VD1742
AENO
MOVR   VD1720, VD1734
AENO
MOVR   VD1724, VD1738
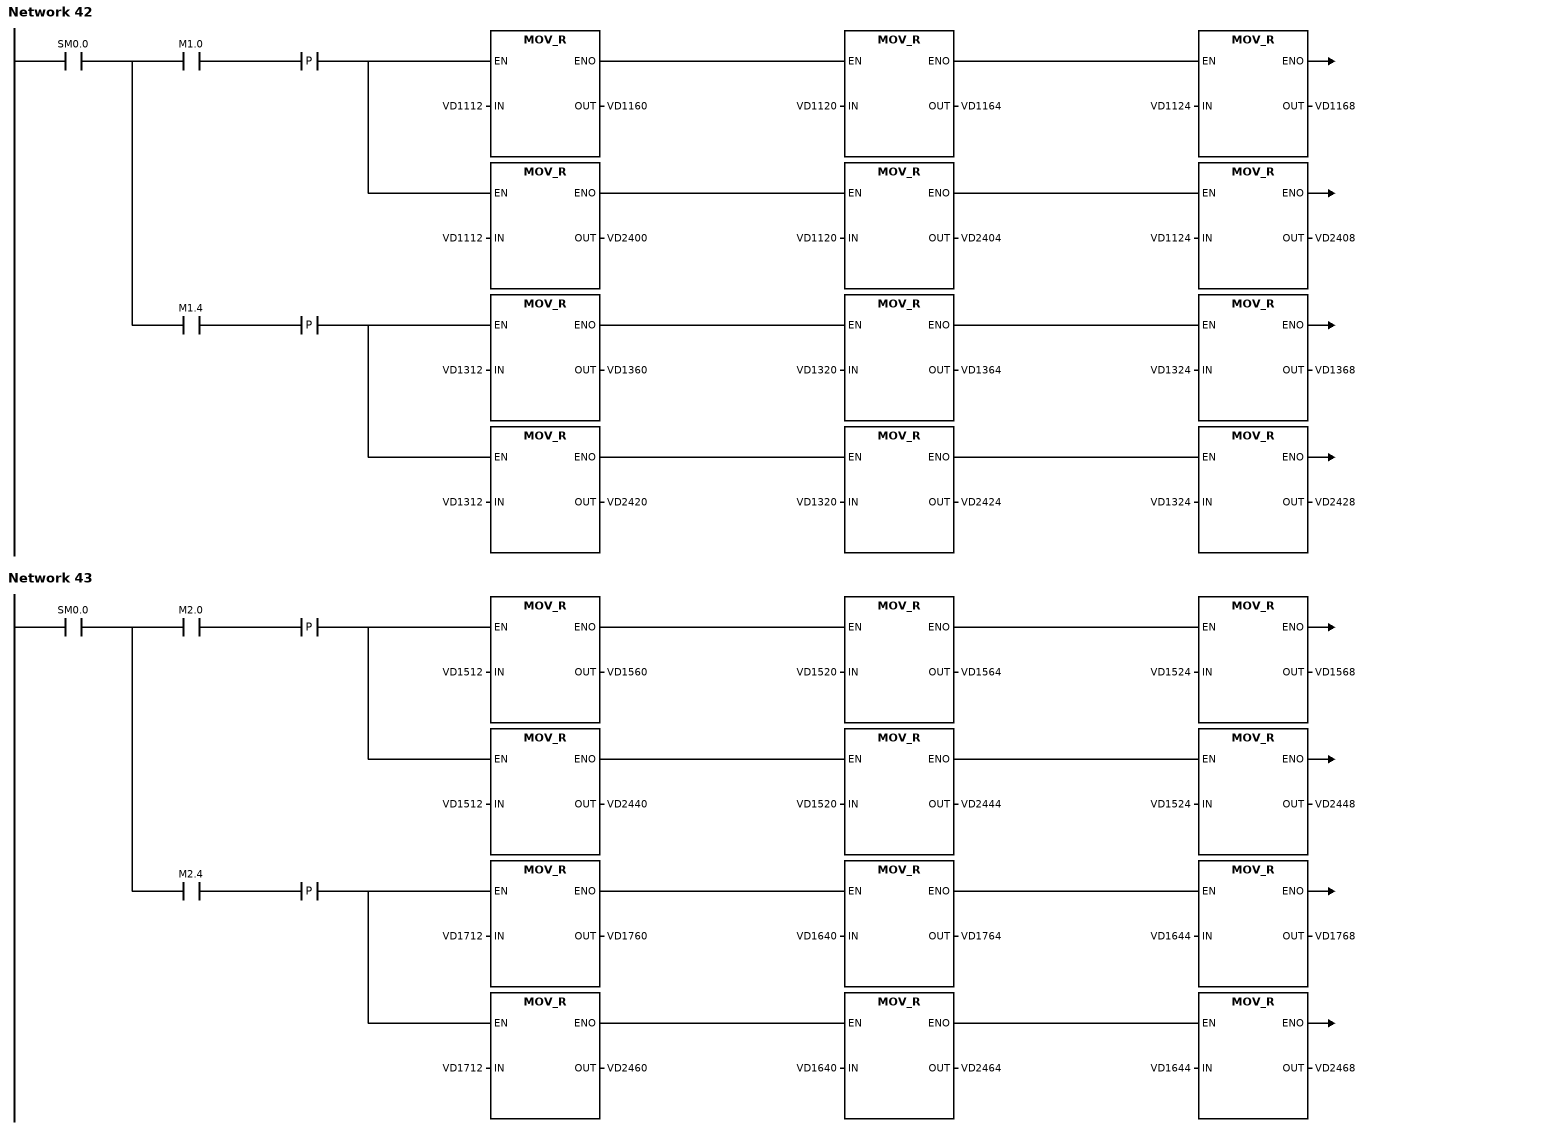
Network 42
LD     SM0.0
LPS
A      M1.0
EU
LPS
MOVR   VD1112, VD1160
AENO
MOVR   VD1120, VD1164
AENO
MOVR   VD1124, VD1168
LPP
MOVR   VD1112, VD2400
AENO
MOVR   VD1120, VD2404
AENO
MOVR   VD1124, VD2408
LPP
A      M1.4
EU
LPS
MOVR   VD1312, VD1360
AENO
MOVR   VD1320, VD1364
AENO
MOVR   VD1324, VD1368
LPP
MOVR   VD1312, VD2420
AENO
MOVR   VD1320, VD2424
AENO
MOVR   VD1324, VD2428
Network 43
LD     SM0.0
LPS
A      M2.0
EU
LPS
MOVR   VD1512, VD1560
AENO
MOVR   VD1520, VD1564
AENO
MOVR   VD1524, VD1568
LPP
MOVR   VD1512, VD2440
AENO
MOVR   VD1520, VD2444
AENO
MOVR   VD1524, VD2448
LPP
A      M2.4
EU
LPS
MOVR   VD1712, VD1760
AENO
MOVR   VD1640, VD1764
AENO
MOVR   VD1644, VD1768
LPP
MOVR   VD1712, VD2460
AENO
MOVR   VD1640, VD2464
AENO
MOVR   VD1644, VD2468
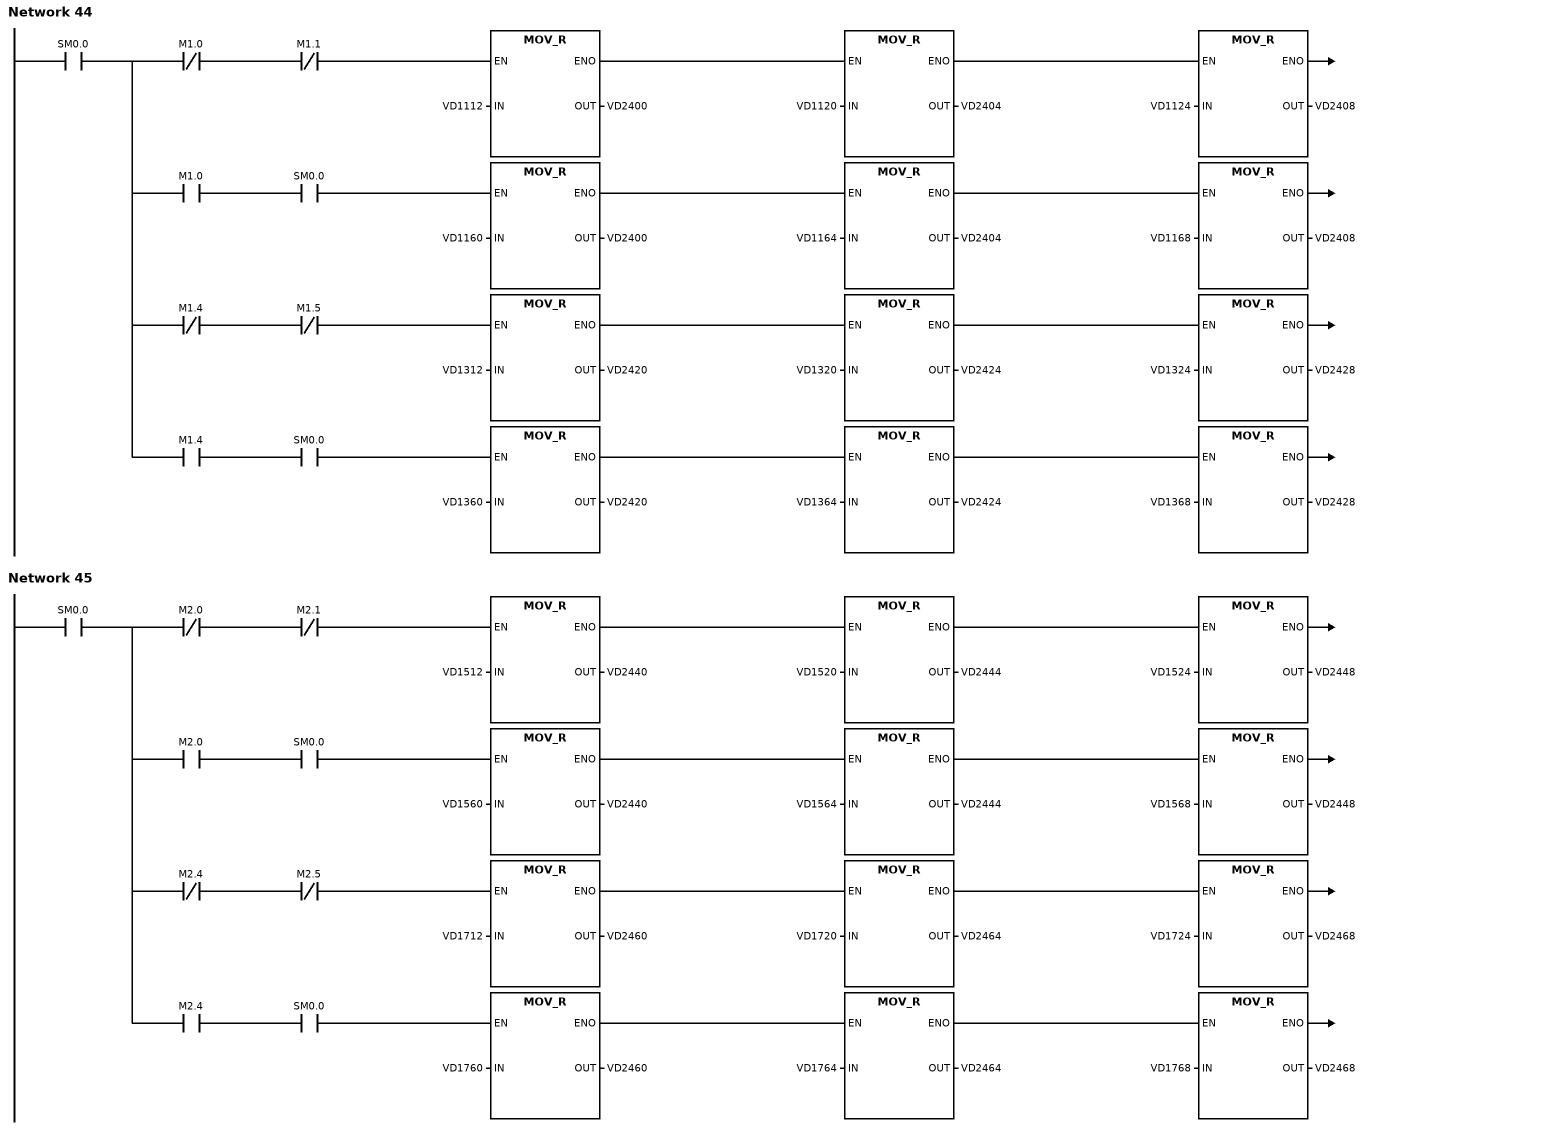
Network 44
LD     SM0.0
LPS
AN     M1.0
AN     M1.1
MOVR   VD1112, VD2400
AENO
MOVR   VD1120, VD2404
AENO
MOVR   VD1124, VD2408
LRD
A      M1.0
A      SM0.0
MOVR   VD1160, VD2400
AENO
MOVR   VD1164, VD2404
AENO
MOVR   VD1168, VD2408
LRD
AN     M1.4
AN     M1.5
MOVR   VD1312, VD2420
AENO
MOVR   VD1320, VD2424
AENO
MOVR   VD1324, VD2428
LPP
A      M1.4
A      SM0.0
MOVR   VD1360, VD2420
AENO
MOVR   VD1364, VD2424
AENO
MOVR   VD1368, VD2428
Network 45
LD     SM0.0
LPS
AN     M2.0
AN     M2.1
MOVR   VD1512, VD2440
AENO
MOVR   VD1520, VD2444
AENO
MOVR   VD1524, VD2448
LRD
A      M2.0
A      SM0.0
MOVR   VD1560, VD2440
AENO
MOVR   VD1564, VD2444
AENO
MOVR   VD1568, VD2448
LRD
AN     M2.4
AN     M2.5
MOVR   VD1712, VD2460
AENO
MOVR   VD1720, VD2464
AENO
MOVR   VD1724, VD2468
LPP
A      M2.4
A      SM0.0
MOVR   VD1760, VD2460
AENO
MOVR   VD1764, VD2464
AENO
MOVR   VD1768, VD2468
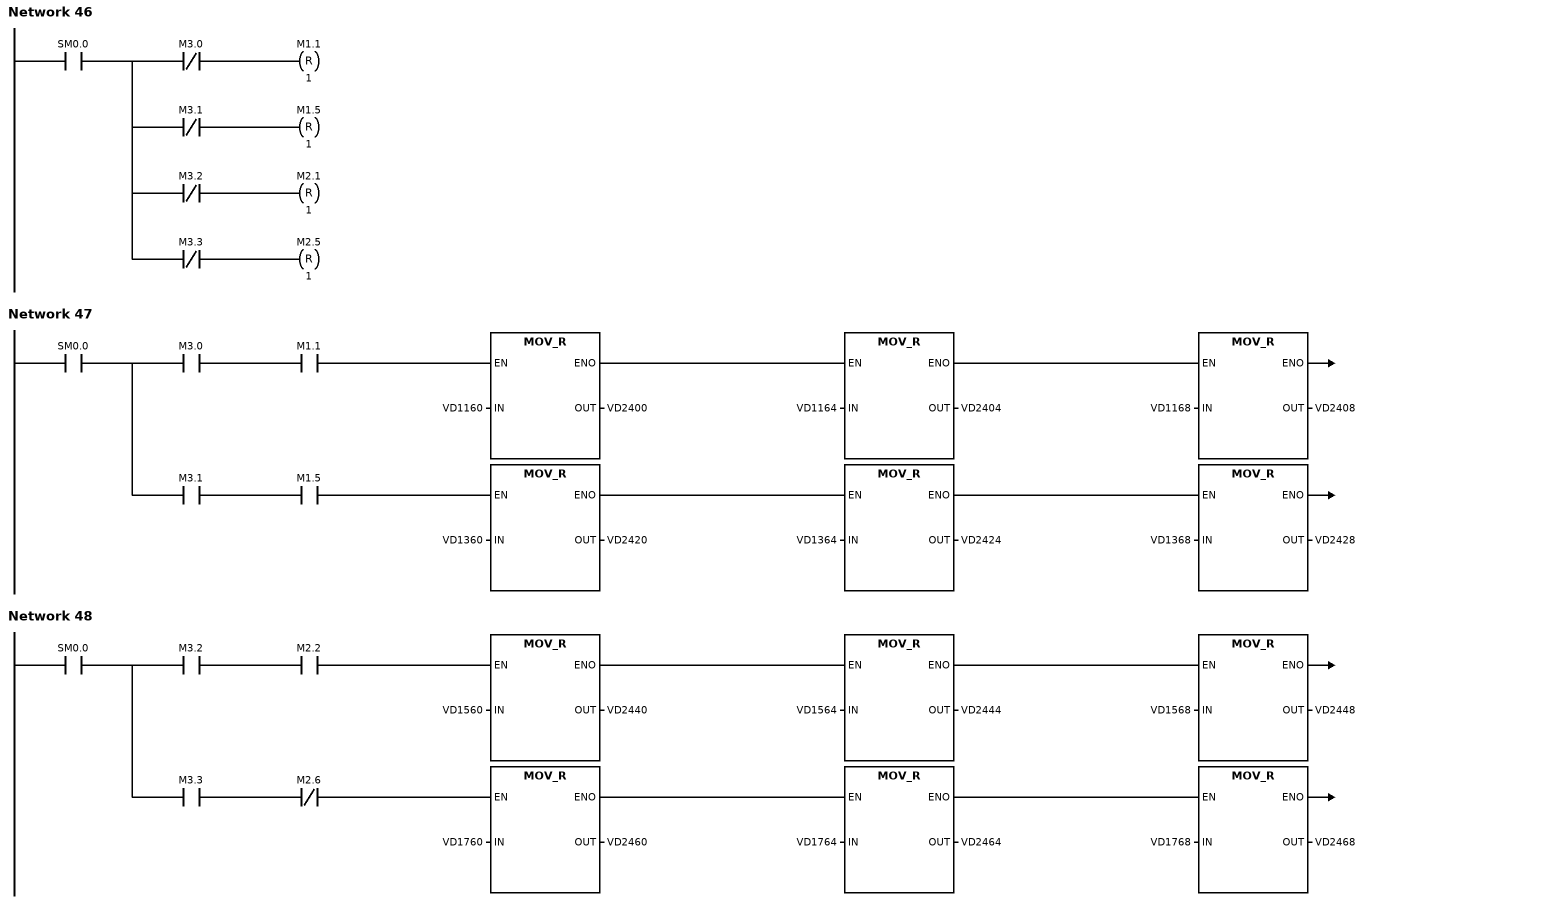
Network 46
LD     SM0.0
LPS
AN     M3.0
R      M1.1, 1
LRD
AN     M3.1
R      M1.5, 1
LRD
AN     M3.2
R      M2.1, 1
LPP
AN     M3.3
R      M2.5, 1
Network 47
LD     SM0.0
LPS
A      M3.0
A      M1.1
MOVR   VD1160, VD2400
AENO
MOVR   VD1164, VD2404
AENO
MOVR   VD1168, VD2408
LPP
A      M3.1
A      M1.5
MOVR   VD1360, VD2420
AENO
MOVR   VD1364, VD2424
AENO
MOVR   VD1368, VD2428
Network 48
LD     SM0.0
LPS
A      M3.2
A      M2.2
MOVR   VD1560, VD2440
AENO
MOVR   VD1564, VD2444
AENO
MOVR   VD1568, VD2448
LPP
A      M3.3
AN     M2.6
MOVR   VD1760, VD2460
AENO
MOVR   VD1764, VD2464
AENO
MOVR   VD1768, VD2468
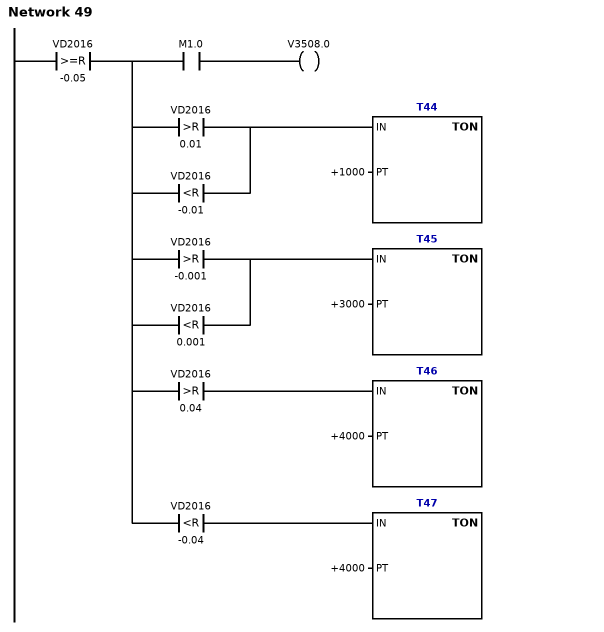
Network 49
LDR>=  VD2016, -0.05
LPS
A      M1.0
=      V3508.0
LRD
LDR>   VD2016, 0.01
OR<    VD2016, -0.01
ALD
TON    T44, +1000
LRD
LDR>   VD2016, -0.001
OR<    VD2016, 0.001
ALD
TON    T45, +3000
LPP
LPS
AR>    VD2016, 0.04
TON    T46, +4000
LPP
AR<    VD2016, -0.04
TON    T47, +4000
